(* Logix 5000 project; controller PHOTON Emulate 5570 rev 30.12; software revision 30.00; part 2 of 2 *)
(* tags used below, declared in another part *)
   PHT_Bit_indxj : DINT;
   PHT_Byte_indxi : DINT;
   PHT_D : DINT;
   PHT_Digest : DINT[60];
   PHT_DIGESTSIZE : DINT;
   PHT_GetByte_BitOffSet : DINT;
   PHT_GetByte_NoOfBits : DINT;
   PHT_GetByte_Res : DINT;
   PHT_Message : DINT[1024];
   PHT_MsgBitLen : DINT;
   PHT_Per_i : DINT;
   PHT_Per_r : DINT;
   PHT_RATEP : DINT;
   PHT_RC : DINT[8,12];
   PHT_round : DINT;
   PHT_S : DINT;
   PHT_SCS_c : DINT;
   PHT_SCS_i : DINT;
   PHT_SCS_index : DINT;
   PHT_SCS_indxi : DINT;
   PHT_SCS_j : DINT;
   PHT_SCS_OS : DINT[8,8];
   PHT_SCS_r : DINT;
   PHT_SCS_v : DINT[2];
   PHT_Squeeze_i : DINT;
   PHT_Squeeze_tmp : DINT;
   PHT_State : DINT[8,8];
   PHT_Table : DINT[8,256,2];
   PHT_Tmp : DINT[2];
   PHT_Ver : DINT;
   PHT_WordToByte_BitOffSet : DINT;
   PHT_WordToByte_i : DINT;
   PHT_WordToByte_NoOfBits : DINT;
   PHT_WordXorByte_BitOffSet : DINT;
   PHT_WordXorByte_i : DINT;
   PHT_WordXorByte_NoOfBits : DINT;
   PHT_WordXorByte_WordOffset : DINT;
   PHT_WriteByte_BitOffset : DINT;
   PHT_WriteByte_LocalFilter : DINT;
   PHT_WriteByte_NoOfBits : DINT;
   PHT_WriteByte_Value : DINT;
   Test_i : DINT;
(* MainProgram, continued *)

   		 PHT_Table[0,139,1]:=31475;
   		 PHT_Table[1,139,0]:=-1469736252;
   		 PHT_Table[1,139,1]:=18301;
   		 PHT_Table[2,139,0]:=-1123298825;
   		 PHT_Table[2,139,1]:=15795;
   		 PHT_Table[3,139,0]:=685799435;
   		 PHT_Table[3,139,1]:=31438;
   		 PHT_Table[4,139,0]:=244012053;
   		 PHT_Table[4,139,1]:=15758;
   		 PHT_Table[5,139,0]:=-1548456453;
   		 PHT_Table[5,139,1]:=62656;
   		 PHT_Table[0,140,0]:=-61122167;
   		 PHT_Table[0,140,1]:=51213;
   		 PHT_Table[1,140,0]:=-1895324903;
   		 PHT_Table[1,140,1]:=44110;
   		 PHT_Table[2,140,0]:=808429162;
   		 PHT_Table[2,140,1]:=25639;
   		 PHT_Table[3,140,0]:=-613714385;
   		 PHT_Table[3,140,1]:=51305;
   		 PHT_Table[4,140,0]:=393988799;
   		 PHT_Table[4,140,1]:=25667;
   		 PHT_Table[5,140,0]:=-1600009789;
   		 PHT_Table[5,140,1]:=35710;
   		 PHT_Table[0,141,0]:=-283086275;
   		 PHT_Table[0,141,1]:=47838;
   		 PHT_Table[1,141,0]:=-874550308;
   		 PHT_Table[1,141,1]:=59147;
   		 PHT_Table[2,141,0]:=-237246728;
   		 PHT_Table[2,141,1]:=23944;
   		 PHT_Table[3,141,0]:=1741793755;
   		 PHT_Table[3,141,1]:=47747;
   		 PHT_Table[4,141,0]:=2037901370;
   		 PHT_Table[4,141,1]:=24021;
   		 PHT_Table[5,141,0]:=272208786;
   		 PHT_Table[5,141,1]:=28666;
   		 PHT_Table[0,142,0]:=1062264297;
   		 PHT_Table[0,142,1]:=13000;
   		 PHT_Table[1,142,0]:=1699180237;
   		 PHT_Table[1,142,1]:=11166;
   		 PHT_Table[2,142,0]:=206414999;
   		 PHT_Table[2,142,1]:=6479;
   		 PHT_Table[3,142,0]:=1885114445;
   		 PHT_Table[3,142,1]:=13009;
   		 PHT_Table[4,142,0]:=1129889641;
   		 PHT_Table[4,142,1]:=6486;
   		 PHT_Table[5,142,0]:=686029174;
   		 PHT_Table[5,142,1]:=25746;
   		 PHT_Table[0,143,0]:=74596581;
   		 PHT_Table[0,143,1]:=59061;
   		 PHT_Table[1,143,0]:=-1286663590;
   		 PHT_Table[1,143,1]:=38276;
   		 PHT_Table[2,143,0]:=-2037747731;
   		 PHT_Table[2,143,1]:=29506;
   		 PHT_Table[3,143,0]:=1190447754;
   		 PHT_Table[3,143,1]:=59078;
   		 PHT_Table[4,143,0]:=-998255563;
   		 PHT_Table[4,143,1]:=29489;
   		 PHT_Table[5,143,0]:=958463749;
   		 PHT_Table[5,143,1]:=55042;
   		 PHT_Table[0,144,0]:=1954349543;
   		 PHT_Table[0,144,1]:=49197;
   		 PHT_Table[1,144,0]:=1673195800;
   		 PHT_Table[1,144,1]:=41078;
   		 PHT_Table[2,144,0]:=1288713999;
   		 PHT_Table[2,144,1]:=24635;
   		 PHT_Table[3,144,0]:=1328665040;
   		 PHT_Table[3,144,1]:=49229;
   		 PHT_Table[4,144,0]:=2013051951;
   		 PHT_Table[4,144,1]:=24667;
   		 PHT_Table[5,144,0]:=-1282539927;
   		 PHT_Table[5,144,1]:=39738;
   		 PHT_Table[0,145,0]:=-1842813959;
   		 PHT_Table[0,145,1]:=6500;
   		 PHT_Table[1,145,0]:=-1079101461;
   		 PHT_Table[1,145,1]:=38991;
   		 PHT_Table[2,145,0]:=111891142;
   		 PHT_Table[2,145,1]:=33194;
   		 PHT_Table[3,145,0]:=942557355;
   		 PHT_Table[3,145,1]:=6629;
   		 PHT_Table[4,145,0]:=-1406348615;
   		 PHT_Table[4,145,1]:=33067;
   		 PHT_Table[5,145,0]:=352121147;
   		 PHT_Table[5,145,1]:=12873;
   		 PHT_Table[0,146,0]:=-1112857175;
   		 PHT_Table[0,146,1]:=40526;
   		 PHT_Table[1,146,0]:=550375765;
   		 PHT_Table[1,146,1]:=53751;
   		 PHT_Table[2,146,0]:=620253640;
   		 PHT_Table[2,146,1]:=20470;
   		 PHT_Table[3,146,0]:=1267719672;
   		 PHT_Table[3,146,1]:=40449;
   		 PHT_Table[4,146,0]:=-762114044;
   		 PHT_Table[4,146,1]:=20409;
   		 PHT_Table[5,146,0]:=-660612775;
   		 PHT_Table[5,146,1]:=10195;
   		 PHT_Table[0,147,0]:=2097713604;
   		 PHT_Table[0,147,1]:=41914;
   		 PHT_Table[1,147,0]:=1953586231;
   		 PHT_Table[1,147,1]:=32580;
   		 PHT_Table[2,147,0]:=-143608770;
   		 PHT_Table[2,147,1]:=56354;
   		 PHT_Table[3,147,0]:=1610604912;
   		 PHT_Table[3,147,1]:=41830;
   		 PHT_Table[4,147,0]:=-715441533;
   		 PHT_Table[4,147,1]:=56574;
   		 PHT_Table[5,147,0]:=80044713;
   		 PHT_Table[5,147,1]:=23987;
   		 PHT_Table[0,148,0]:=1748556394;
   		 PHT_Table[0,148,1]:=17419;
   		 PHT_Table[1,148,0]:=1464635269;
   		 PHT_Table[1,148,1]:=26311;
   		 PHT_Table[2,148,0]:=-213179974;
   		 PHT_Table[2,148,1]:=8942;
   		 PHT_Table[3,148,0]:=-2033479349;
   		 PHT_Table[3,148,1]:=17449;
   		 PHT_Table[4,148,0]:=496674468;
   		 PHT_Table[4,148,1]:=8908;
   		 PHT_Table[5,148,0]:=476919154;
   		 PHT_Table[5,148,1]:=34868;
   		 PHT_Table[0,149,0]:=1668573878;
   		 PHT_Table[0,149,1]:=21579;
   		 PHT_Table[1,149,0]:=-1808979065;
   		 PHT_Table[1,149,1]:=32439;
   		 PHT_Table[2,149,0]:=195958896;
   		 PHT_Table[2,149,1]:=10966;
   		 PHT_Table[3,149,0]:=-1249917778;
   		 PHT_Table[3,149,1]:=21601;
   		 PHT_Table[4,149,0]:=-577811809;
   		 PHT_Table[4,149,1]:=11004;
   		 PHT_Table[5,149,0]:=976575293;
   		 PHT_Table[5,149,1]:=43196;
   		 PHT_Table[0,150,0]:=-1506505012;
   		 PHT_Table[0,150,1]:=15340;
   		 PHT_Table[1,150,0]:=428408100;
   		 PHT_Table[1,150,1]:=43937;
   		 PHT_Table[2,150,0]:=-234631269;
   		 PHT_Table[2,150,1]:=37085;
   		 PHT_Table[3,150,0]:=2076609795;
   		 PHT_Table[3,150,1]:=15228;
   		 PHT_Table[4,150,0]:=794919403;
   		 PHT_Table[4,150,1]:=36941;
   		 PHT_Table[5,150,0]:=440886786;
   		 PHT_Table[5,150,1]:=30291;
   		 PHT_Table[0,151,0]:=-1142929997;
   		 PHT_Table[0,151,1]:=2860;
   		 PHT_Table[1,151,0]:=1194002978;
   		 PHT_Table[1,151,1]:=33585;
   		 PHT_Table[2,151,0]:=-516455202;
   		 PHT_Table[2,151,1]:=34965;
   		 PHT_Table[3,151,0]:=771846711;
   		 PHT_Table[3,151,1]:=2980;
   		 PHT_Table[4,151,0]:=1952362150;
   		 PHT_Table[4,151,1]:=34845;
   		 PHT_Table[5,151,0]:=1890571475;
   		 PHT_Table[5,151,1]:=5840;
   		 PHT_Table[0,152,0]:=-1805417501;
   		 PHT_Table[0,152,1]:=35846;
   		 PHT_Table[1,152,0]:=-666162020;
   		 PHT_Table[1,152,1]:=51849;
   		 PHT_Table[2,152,0]:=-1016821808;
   		 PHT_Table[2,152,1]:=18121;
   		 PHT_Table[3,152,0]:=1570826084;
   		 PHT_Table[3,152,1]:=35904;
   		 PHT_Table[4,152,0]:=182545435;
   		 PHT_Table[4,152,1]:=18063;
   		 PHT_Table[5,152,0]:=-1127416655;
   		 PHT_Table[5,152,1]:=842;
   		 PHT_Table[0,153,0]:=61353997;
   		 PHT_Table[0,153,1]:=50993;
   		 PHT_Table[1,153,0]:=-1090551626;
   		 PHT_Table[1,153,1]:=10595;
   		 PHT_Table[2,153,0]:=-269818101;
   		 PHT_Table[2,153,1]:=61116;
   		 PHT_Table[3,153,0]:=-1085809942;
   		 PHT_Table[3,153,1]:=51167;
   		 PHT_Table[4,153,0]:=1407934289;
   		 PHT_Table[4,153,1]:=61010;
   		 PHT_Table[5,153,0]:=1410894661;
   		 PHT_Table[5,153,1]:=38284;
   		 PHT_Table[0,154,0]:=-2125215667;
   		 PHT_Table[0,154,1]:=27575;
   		 PHT_Table[1,154,0]:=-76087506;
   		 PHT_Table[1,154,1]:=54026;
   		 PHT_Table[2,154,0]:=-950070700;
   		 PHT_Table[2,154,1]:=47109;
   		 PHT_Table[3,154,0]:=-2070636705;
   		 PHT_Table[3,154,1]:=27407;
   		 PHT_Table[4,154,0]:=-1038028740;
   		 PHT_Table[4,154,1]:=47293;
   		 PHT_Table[5,154,0]:=-1536906390;
   		 PHT_Table[5,154,1]:=54989;
   		 PHT_Table[0,155,0]:=-1631706163;
   		 PHT_Table[0,155,1]:=10400;
   		 PHT_Table[1,155,0]:=1904148741;
   		 PHT_Table[1,155,1]:=15576;
   		 PHT_Table[2,155,0]:=-1758534678;
   		 PHT_Table[2,155,1]:=5228;
   		 PHT_Table[3,155,0]:=-232190674;
   		 PHT_Table[3,155,1]:=10420;
   		 PHT_Table[4,155,0]:=-72501786;
   		 PHT_Table[4,155,1]:=5240;
   		 PHT_Table[5,155,0]:=1604119348;
   		 PHT_Table[5,155,1]:=20559;
   		 PHT_Table[0,156,0]:=958119411;
   		 PHT_Table[0,156,1]:=42922;
   		 PHT_Table[1,156,0]:=44201402;
   		 PHT_Table[1,156,1]:=31064;
   		 PHT_Table[2,156,0]:=-914198143;
   		 PHT_Table[2,156,1]:=56876;
   		 PHT_Table[3,156,0]:=366100354;
   		 PHT_Table[3,156,1]:=42868;
   		 PHT_Table[4,156,0]:=-443219509;
   		 PHT_Table[4,156,1]:=57074;
   		 PHT_Table[5,156,0]:=-2133592836;
   		 PHT_Table[5,156,1]:=21905;
   		 PHT_Table[0,157,0]:=-1984477028;
   		 PHT_Table[0,157,1]:=48326;
   		 PHT_Table[1,157,0]:=-2031559782;
   		 PHT_Table[1,157,1]:=57881;
   		 PHT_Table[2,157,0]:=-800011115;
   		 PHT_Table[2,157,1]:=24193;
   		 PHT_Table[3,157,0]:=140974160;
   		 PHT_Table[3,157,1]:=48280;
   		 PHT_Table[4,157,0]:=1373520726;
   		 PHT_Table[4,157,1]:=24287;
   		 PHT_Table[5,157,0]:=-702263712;
   		 PHT_Table[5,157,1]:=25545;
   		 PHT_Table[0,158,0]:=1843104381;
   		 PHT_Table[0,158,1]:=5720;
   		 PHT_Table[1,158,0]:=-1906961340;
   		 PHT_Table[1,158,1]:=7522;
   		 PHT_Table[2,158,0]:=-647097433;
   		 PHT_Table[2,158,1]:=2865;
   		 PHT_Table[3,158,0]:=1543693422;
   		 PHT_Table[3,158,1]:=5715;
   		 PHT_Table[4,158,0]:=-390314153;
   		 PHT_Table[4,158,1]:=2874;
   		 PHT_Table[5,158,0]:=-532302915;
   		 PHT_Table[5,158,1]:=11451;
   		 PHT_Table[0,159,0]:=-1816530165;
   		 PHT_Table[0,159,1]:=44418;
   		 PHT_Table[1,159,0]:=-704922000;
   		 PHT_Table[1,159,1]:=30318;
   		 PHT_Table[2,159,0]:=-1442574538;
   		 PHT_Table[2,159,1]:=56119;
   		 PHT_Table[3,159,0]:=-1542195452;
   		 PHT_Table[3,159,1]:=44377;
   		 PHT_Table[4,159,0]:=-1653217409;
   		 PHT_Table[4,159,1]:=56300;
   		 PHT_Table[5,159,0]:=-772503311;
   		 PHT_Table[5,159,1]:=16836;
   		 PHT_Table[0,160,0]:=-992873336;
   		 PHT_Table[0,160,1]:=56129;
   		 PHT_Table[1,160,0]:=-403677384;
   		 PHT_Table[1,160,1]:=15159;
   		 PHT_Table[2,160,0]:=1426229787;
   		 PHT_Table[2,160,1]:=57494;
   		 PHT_Table[3,160,0]:=1384445442;
   		 PHT_Table[3,160,1]:=56225;
   		 PHT_Table[4,160,0]:=-1011351886;
   		 PHT_Table[4,160,1]:=57462;
   		 PHT_Table[5,160,0]:=-444971787;
   		 PHT_Table[5,160,1]:=44386;
   		 PHT_Table[0,161,0]:=2124456393;
   		 PHT_Table[0,161,1]:=25739;
   		 PHT_Table[1,161,0]:=-896607103;
   		 PHT_Table[1,161,1]:=22055;
   		 PHT_Table[2,161,0]:=412767029;
   		 PHT_Table[2,161,1]:=12958;
   		 PHT_Table[3,161,0]:=-524797030;
   		 PHT_Table[3,161,1]:=25785;
   		 PHT_Table[4,161,0]:=-2035259950;
   		 PHT_Table[4,161,1]:=12972;
   		 PHT_Table[5,161,0]:=1356720620;
   		 PHT_Table[5,161,1]:=51263;
   		 PHT_Table[0,162,0]:=1978405141;
   		 PHT_Table[0,162,1]:=29899;
   		 PHT_Table[1,162,0]:=166688899;
   		 PHT_Table[1,162,1]:=20055;
   		 PHT_Table[2,162,0]:=-528520449;
   		 PHT_Table[2,162,1]:=15014;
   		 PHT_Table[3,162,0]:=-754160001;
   		 PHT_Table[3,162,1]:=29937;
   		 PHT_Table[4,162,0]:=1185253865;
   		 PHT_Table[4,162,1]:=15004;
   		 PHT_Table[5,162,0]:=1988462499;
   		 PHT_Table[5,162,1]:=59575;
   		 PHT_Table[0,163,0]:=1331666155;
   		 PHT_Table[0,163,1]:=5200;
   		 PHT_Table[1,163,0]:=-1246589553;
   		 PHT_Table[1,163,1]:=7788;
   		 PHT_Table[2,163,0]:=-971506571;
   		 PHT_Table[2,163,1]:=2614;
   		 PHT_Table[3,163,0]:=2040105751;
   		 PHT_Table[3,163,1]:=5210;
   		 PHT_Table[4,163,0]:=-254027917;
   		 PHT_Table[4,163,1]:=2620;
   		 PHT_Table[5,163,0]:=-1571882982;
   		 PHT_Table[5,163,1]:=10410;
   		 PHT_Table[0,164,0]:=1906201072;
   		 PHT_Table[0,164,1]:=37502;
   		 PHT_Table[1,164,0]:=-1163892007;
   		 PHT_Table[1,164,1]:=56275;
   		 PHT_Table[2,164,0]:=1727333650;
   		 PHT_Table[2,164,1]:=18916;
   		 PHT_Table[3,164,0]:=-1778866955;
   		 PHT_Table[3,164,1]:=37431;
   		 PHT_Table[4,164,0]:=-2099618340;
   		 PHT_Table[4,164,1]:=18861;
   		 PHT_Table[5,164,0]:=1336244390;
   		 PHT_Table[5,164,1]:=16309;
   		 PHT_Table[0,165,0]:=-868912039;
   		 PHT_Table[0,165,1]:=3120;
   		 PHT_Table[1,165,0]:=-1704035444;
   		 PHT_Table[1,165,1]:=2596;
   		 PHT_Table[2,165,0]:=1108169946;
   		 PHT_Table[2,165,1]:=1554;
   		 PHT_Table[3,165,0]:=-562595571;
   		 PHT_Table[3,165,1]:=3126;
   		 PHT_Table[4,165,0]:=1346981336;
   		 PHT_Table[4,165,1]:=1556;
   		 PHT_Table[5,165,0]:=-1757765121;
   		 PHT_Table[5,165,1]:=6246;
   		 PHT_Table[0,166,0]:=-1542607309;
   		 PHT_Table[0,166,1]:=18491;
   		 PHT_Table[1,166,0]:=-853347319;
   		 PHT_Table[1,166,1]:=27875;
   		 PHT_Table[2,166,0]:=-1320782496;
   		 PHT_Table[2,166,1]:=9468;
   		 PHT_Table[3,166,0]:=1488775238;
   		 PHT_Table[3,166,1]:=18463;
   		 PHT_Table[4,166,0]:=1305734012;
   		 PHT_Table[4,166,1]:=9432;
   		 PHT_Table[5,166,0]:=-1957194611;
   		 PHT_Table[5,166,1]:=36946;
   		 PHT_Table[0,167,0]:=-844864341;
   		 PHT_Table[0,167,1]:=47318;
   		 PHT_Table[1,167,0]:=-264506857;
   		 PHT_Table[1,167,1]:=58373;
   		 PHT_Table[2,167,0]:=-291370710;
   		 PHT_Table[2,167,1]:=23695;
   		 PHT_Table[3,167,0]:=1112196770;
   		 PHT_Table[3,167,1]:=47242;
   		 PHT_Table[4,167,0]:=1628469278;
   		 PHT_Table[4,167,1]:=23763;
   		 PHT_Table[5,167,0]:=1379063861;
   		 PHT_Table[5,167,1]:=27627;
   		 PHT_Table[0,168,0]:=-1394004254;
   		 PHT_Table[0,168,1]:=40778;
   		 PHT_Table[1,168,0]:=-1329803075;
   		 PHT_Table[1,168,1]:=24048;
   		 PHT_Table[2,168,0]:=-1505121375;
   		 PHT_Table[2,168,1]:=49784;
   		 PHT_Table[3,168,0]:=-732993719;
   		 PHT_Table[3,168,1]:=40840;
   		 PHT_Table[4,168,0]:=-567453674;
   		 PHT_Table[4,168,1]:=49850;
   		 PHT_Table[5,168,0]:=-115904121;
   		 PHT_Table[5,168,1]:=9558;
   		 PHT_Table[0,169,0]:=-1728756777;
   		 PHT_Table[0,169,1]:=48578;
   		 PHT_Table[1,169,0]:=379198066;
   		 PHT_Table[1,169,1]:=28190;
   		 PHT_Table[2,169,0]:=1390491388;
   		 PHT_Table[2,169,1]:=54031;
   		 PHT_Table[3,169,0]:=-1750621471;
   		 PHT_Table[3,169,1]:=48401;
   		 PHT_Table[4,169,0]:=1566575428;
   		 PHT_Table[4,169,1]:=54236;
   		 PHT_Table[5,169,0]:=-139663682;
   		 PHT_Table[5,169,1]:=24908;
   		 PHT_Table[0,170,0]:=535686016;
   		 PHT_Table[0,170,1]:=17175;
   		 PHT_Table[1,170,0]:=-1979056597;
   		 PHT_Table[1,170,1]:=61394;
   		 PHT_Table[2,170,0]:=1349644734;
   		 PHT_Table[2,170,1]:=44137;
   		 PHT_Table[3,170,0]:=1992137329;
   		 PHT_Table[3,170,1]:=17339;
   		 PHT_Table[4,170,0]:=965559770;
   		 PHT_Table[4,170,1]:=44229;
   		 PHT_Table[5,170,0]:=-67616674;
   		 PHT_Table[5,170,1]:=34434;
   		 PHT_Table[0,171,0]:=812527056;
   		 PHT_Table[0,171,1]:=50237;
   		 PHT_Table[1,171,0]:=359258261;
   		 PHT_Table[1,171,1]:=42602;
   		 PHT_Table[2,171,0]:=1914892976;
   		 PHT_Table[2,171,1]:=25141;
   		 PHT_Table[3,171,0]:=85724962;
   		 PHT_Table[3,171,1]:=50271;
   		 PHT_Table[4,171,0]:=1194493799;
   		 PHT_Table[4,171,1]:=25175;
   		 PHT_Table[5,171,0]:=932931644;
   		 PHT_Table[5,171,1]:=37656;
   		 PHT_Table[0,172,0]:=-2068801446;
   		 PHT_Table[0,172,1]:=14820;
   		 PHT_Table[1,172,0]:=577529071;
   		 PHT_Table[1,172,1]:=43183;
   		 PHT_Table[2,172,0]:=-310763447;
   		 PHT_Table[2,172,1]:=37338;
   		 PHT_Table[3,172,0]:=1583211130;
   		 PHT_Table[3,172,1]:=14709;
   		 PHT_Table[4,172,0]:=923144655;
   		 PHT_Table[4,172,1]:=37195;
   		 PHT_Table[5,172,0]:=1481387429;
   		 PHT_Table[5,172,1]:=29250;
   		 PHT_Table[0,173,0]:=211206196;
   		 PHT_Table[0,173,1]:=12740;
   		 PHT_Table[1,173,0]:=-825149714;
   		 PHT_Table[1,173,1]:=42135;
   		 PHT_Table[2,173,0]:=-1853509332;
   		 PHT_Table[2,173,1]:=38342;
   		 PHT_Table[3,173,0]:=-905493115;
   		 PHT_Table[3,173,1]:=12625;
   		 PHT_Table[4,173,0]:=1468098399;
   		 PHT_Table[4,173,1]:=38227;
   		 PHT_Table[5,173,0]:=1264589327;
   		 PHT_Table[5,173,1]:=25094;
   		 PHT_Table[0,174,0]:=1291300070;
   		 PHT_Table[0,174,1]:=54113;
   		 PHT_Table[1,174,0]:=189599033;
   		 PHT_Table[1,174,1]:=14095;
   		 PHT_Table[2,174,0]:=704453502;
   		 PHT_Table[2,174,1]:=58506;
   		 PHT_Table[3,174,0]:=-958508547;
   		 PHT_Table[3,174,1]:=54149;
   		 PHT_Table[4,174,0]:=-1557100510;
   		 PHT_Table[4,174,1]:=58478;
   		 PHT_Table[5,174,0]:=-162106529;
   		 PHT_Table[5,174,1]:=48422;
   		 PHT_Table[0,175,0]:=1261296654;
   		 PHT_Table[0,175,1]:=62181;
   		 PHT_Table[1,175,0]:=117284821;
   		 PHT_Table[1,175,1]:=35816;
   		 PHT_Table[2,175,0]:=1084068760;
   		 PHT_Table[2,175,1]:=31092;
   		 PHT_Table[3,175,0]:=1064124829;
   		 PHT_Table[3,175,1]:=62108;
   		 PHT_Table[4,175,0]:=883163974;
   		 PHT_Table[4,175,1]:=30989;
   		 PHT_Table[5,175,0]:=-1687288033;
   		 PHT_Table[5,175,1]:=65448;
   		 PHT_Table[0,176,0]:=710972999;
   		 PHT_Table[0,176,1]:=54649;
   		 PHT_Table[1,176,0]:=1182449023;
   		 PHT_Table[1,176,1]:=12829;
   		 PHT_Table[2,176,0]:=141963539;
   		 PHT_Table[2,176,1]:=59267;
   		 PHT_Table[3,176,0]:=-1452744586;
   		 PHT_Table[3,176,1]:=54686;
   		 PHT_Table[4,176,0]:=-1952898226;
   		 PHT_Table[4,176,1]:=59236;
   		 PHT_Table[5,176,0]:=810266285;
   		 PHT_Table[5,176,1]:=45333;
   		 PHT_Table[0,177,0]:=-474566135;
   		 PHT_Table[0,177,1]:=35610;
   		 PHT_Table[1,177,0]:=84827442;
   		 PHT_Table[1,177,1]:=17308;
   		 PHT_Table[2,177,0]:=1616795604;
   		 PHT_Table[2,177,1]:=51278;
   		 PHT_Table[3,177,0]:=-1378423714;
   		 PHT_Table[3,177,1]:=35794;
   		 PHT_Table[4,177,0]:=787910501;
   		 PHT_Table[4,177,1]:=51334;
   		 PHT_Table[5,177,0]:=1532594589;
   		 PHT_Table[5,177,1]:=3580;
   		 PHT_Table[0,178,0]:=-738005199;
   		 PHT_Table[0,178,1]:=28323;
   		 PHT_Table[1,178,0]:=500635467;
   		 PHT_Table[1,178,1]:=22801;
   		 PHT_Table[2,178,0]:=2065444226;
   		 PHT_Table[2,178,1]:=14213;
   		 PHT_Table[3,178,0]:=1366946588;
   		 PHT_Table[3,178,1]:=28308;
   		 PHT_Table[4,178,0]:=-28277914;
   		 PHT_Table[4,178,1]:=14258;
   		 PHT_Table[5,178,0]:=33199585;
   		 PHT_Table[5,178,1]:=56426;
   		 PHT_Table[0,179,0]:=-711721021;
   		 PHT_Table[0,179,1]:=55877;
   		 PHT_Table[1,179,0]:=2005049040;
   		 PHT_Table[1,179,1]:=46896;
   		 PHT_Table[2,179,0]:=-676106126;
   		 PHT_Table[2,179,1]:=27928;
   		 PHT_Table[3,179,0]:=-851161933;
   		 PHT_Table[3,179,1]:=55848;
   		 PHT_Table[4,179,0]:=-821447008;
   		 PHT_Table[4,179,1]:=28021;
   		 PHT_Table[5,179,0]:=-990712789;
   		 PHT_Table[5,179,1]:=45031;
   		 PHT_Table[0,180,0]:=289540939;
   		 PHT_Table[0,180,1]:=260;
   		 PHT_Table[1,180,0]:=-1871527448;
   		 PHT_Table[1,180,1]:=35847;
   		 PHT_Table[2,180,0]:=-2102265239;
   		 PHT_Table[2,180,1]:=36238;
   		 PHT_Table[3,180,0]:=-1614759247;
   		 PHT_Table[3,180,1]:=393;
   		 PHT_Table[4,180,0]:=213796882;
   		 PHT_Table[4,180,1]:=36099;
   		 PHT_Table[5,180,0]:=562604254;
   		 PHT_Table[5,180,1]:=645;
   		 PHT_Table[0,181,0]:=1421883278;
   		 PHT_Table[0,181,1]:=45554;
   		 PHT_Table[1,181,0]:=-1930141186;
   		 PHT_Table[1,181,1]:=25658;
   		 PHT_Table[2,181,0]:=283927078;
   		 PHT_Table[2,181,1]:=54557;
   		 PHT_Table[3,181,0]:=1238424556;
   		 PHT_Table[3,181,1]:=45351;
   		 PHT_Table[4,181,0]:=220808860;
   		 PHT_Table[4,181,1]:=54728;
   		 PHT_Table[5,181,0]:=1620461377;
   		 PHT_Table[5,181,1]:=31018;
   		 PHT_Table[0,182,0]:=-1624296641;
   		 PHT_Table[0,182,1]:=40006;
   		 PHT_Table[1,182,0]:=455772318;
   		 PHT_Table[1,182,1]:=54009;
   		 PHT_Table[2,182,0]:=998358554;
   		 PHT_Table[2,182,1]:=20209;
   		 PHT_Table[3,182,0]:=1846850177;
   		 PHT_Table[3,182,1]:=39944;
   		 PHT_Table[4,182,0]:=-889946080;
   		 PHT_Table[4,182,1]:=20159;
   		 PHT_Table[5,182,0]:=-1701539074;
   		 PHT_Table[5,182,1]:=9154;
   		 PHT_Table[0,183,0]:=-1253071496;
   		 PHT_Table[0,183,1]:=18751;
   		 PHT_Table[1,183,0]:=1565537761;
   		 PHT_Table[1,183,1]:=57572;
   		 PHT_Table[2,183,0]:=871862025;
   		 PHT_Table[2,183,1]:=43378;
   		 PHT_Table[3,183,0]:=-948153609;
   		 PHT_Table[3,183,1]:=18838;
   		 PHT_Table[4,183,0]:=1097704302;
   		 PHT_Table[4,183,1]:=43483;
   		 PHT_Table[5,183,0]:=-1428210605;
   		 PHT_Table[5,183,1]:=37591;
   		 PHT_Table[0,184,0]:=-149427883;
   		 PHT_Table[0,184,1]:=55373;
   		 PHT_Table[1,184,0]:=1281754907;
   		 PHT_Table[1,184,1]:=46142;
   		 PHT_Table[2,184,0]:=-926244960;
   		 PHT_Table[2,184,1]:=27679;
   		 PHT_Table[3,184,0]:=-388029494;
   		 PHT_Table[3,184,1]:=55329;
   		 PHT_Table[4,184,0]:=-680647036;
   		 PHT_Table[4,184,1]:=27763;
   		 PHT_Table[5,184,0]:=-2030458996;
   		 PHT_Table[5,184,1]:=44022;
   		 PHT_Table[0,185,0]:=-2097416128;
   		 PHT_Table[0,185,1]:=44166;
   		 PHT_Table[1,185,0]:=1166639000;
   		 PHT_Table[1,185,1]:=64105;
   		 PHT_Table[2,185,0]:=683013471;
   		 PHT_Table[2,185,1]:=22201;
   		 PHT_Table[3,185,0]:=1003703733;
   		 PHT_Table[3,185,1]:=44240;
   		 PHT_Table[4,185,0]:=-1848922259;
   		 PHT_Table[4,185,1]:=22255;
   		 PHT_Table[5,185,0]:=-260300753;
   		 PHT_Table[5,185,1]:=17217;
   		 PHT_Table[0,186,0]:=1517279045;
   		 PHT_Table[0,186,1]:=62433;
   		 PHT_Table[1,186,0]:=-1768989123;
   		 PHT_Table[1,186,1]:=2031;
   		 PHT_Table[2,186,0]:=-1037276687;
   		 PHT_Table[2,186,1]:=62714;
   		 PHT_Table[3,186,0]:=-1599210708;
   		 PHT_Table[3,186,1]:=62229;
   		 PHT_Table[4,186,0]:=941247316;
   		 PHT_Table[4,186,1]:=62478;
   		 PHT_Table[5,186,0]:=-1159286847;
   		 PHT_Table[5,186,1]:=64813;
   		 PHT_Table[0,187,0]:=-1953601437;
   		 PHT_Table[0,187,1]:=53009;
   		 PHT_Table[1,187,0]:=1380111031;
   		 PHT_Table[1,187,1]:=9563;
   		 PHT_Table[2,187,0]:=-1827309970;
   		 PHT_Table[2,187,1]:=60064;
   		 PHT_Table[3,187,0]:=723352853;
   		 PHT_Table[3,187,1]:=53243;
   		 PHT_Table[4,187,0]:=862726593;
   		 PHT_Table[4,187,1]:=59978;
   		 PHT_Table[5,187,0]:=1194638575;
   		 PHT_Table[5,187,1]:=34248;
   		 PHT_Table[0,188,0]:=-555790561;
   		 PHT_Table[0,188,1]:=51717;
   		 PHT_Table[1,188,0]:=-1260176686;
   		 PHT_Table[1,188,1]:=44864;
   		 PHT_Table[2,188,0]:=794184120;
   		 PHT_Table[2,188,1]:=25888;
   		 PHT_Table[3,188,0]:=-17819306;
   		 PHT_Table[3,188,1]:=51808;
   		 PHT_Table[4,188,0]:=253516443;
   		 PHT_Table[4,188,1]:=25925;
   		 PHT_Table[5,188,0]:=-492141980;
   		 PHT_Table[5,188,1]:=36719;
   		 PHT_Table[0,189,0]:=767223471;
   		 PHT_Table[0,189,1]:=62717;
   		 PHT_Table[1,189,0]:=1271541651;
   		 PHT_Table[1,189,1]:=36602;
   		 PHT_Table[2,189,0]:=1628879349;
   		 PHT_Table[2,189,1]:=31357;
   		 PHT_Table[3,189,0]:=1356591126;
   		 PHT_Table[3,189,1]:=62599;
   		 PHT_Table[4,189,0]:=470657066;
   		 PHT_Table[4,189,1]:=31239;
   		 PHT_Table[5,189,0]:=1567873773;
   		 PHT_Table[5,189,1]:=62363;
   		 PHT_Table[0,190,0]:=1543423927;
   		 PHT_Table[0,190,1]:=18183;
   		 PHT_Table[1,190,0]:=-52766810;
   		 PHT_Table[1,190,1]:=59854;
   		 PHT_Table[2,190,0]:=1854092289;
   		 PHT_Table[2,190,1]:=44647;
   		 PHT_Table[3,190,0]:=1016087683;
   		 PHT_Table[3,190,1]:=18345;
   		 PHT_Table[4,190,0]:=155418258;
   		 PHT_Table[4,190,1]:=44745;
   		 PHT_Table[5,190,0]:=2146358795;
   		 PHT_Table[5,190,1]:=36512;
   		 PHT_Table[0,191,0]:=189575388;
   		 PHT_Table[0,191,1]:=4160;
   		 PHT_Table[1,191,0]:=-1017011198;
   		 PHT_Table[1,191,1]:=6256;
   		 PHT_Table[2,191,0]:=-119195190;
   		 PHT_Table[2,191,1]:=2104;
   		 PHT_Table[3,191,0]:=867456485;
   		 PHT_Table[3,191,1]:=4168;
   		 PHT_Table[4,191,0]:=-1072305093;
   		 PHT_Table[4,191,1]:=2096;
   		 PHT_Table[5,191,0]:=643329615;
   		 PHT_Table[5,191,1]:=8328;
   		 PHT_Table[0,192,0]:=-985602950;
   		 PHT_Table[0,192,1]:=28583;
   		 PHT_Table[1,192,0]:=-1918511453;
   		 PHT_Table[1,192,1]:=54550;
   		 PHT_Table[2,192,0]:=-106047509;
   		 PHT_Table[2,192,1]:=47627;
   		 PHT_Table[3,192,0]:=-826717779;
   		 PHT_Table[3,192,1]:=28445;
   		 PHT_Table[4,192,0]:=-219231372;
   		 PHT_Table[4,192,1]:=47793;
   		 PHT_Table[5,192,0]:=544357695;
   		 PHT_Table[5,192,1]:=57071;
   		 PHT_Table[0,193,0]:=1772735128;
   		 PHT_Table[0,193,1]:=61677;
   		 PHT_Table[1,193,0]:=1025050142;
   		 PHT_Table[1,193,1]:=35046;
   		 PHT_Table[2,193,0]:=1608809546;
   		 PHT_Table[2,193,1]:=30835;
   		 PHT_Table[3,193,0]:=452341476;
   		 PHT_Table[3,193,1]:=61589;
   		 PHT_Table[4,193,0]:=751014754;
   		 PHT_Table[4,193,1]:=30731;
   		 PHT_Table[5,193,0]:=-647672648;
   		 PHT_Table[5,193,1]:=64441;
   		 PHT_Table[0,194,0]:=-2037794651;
   		 PHT_Table[0,194,1]:=18995;
   		 PHT_Table[1,194,0]:=-154767934;
   		 PHT_Table[1,194,1]:=28653;
   		 PHT_Table[2,194,0]:=-1371563342;
   		 PHT_Table[2,194,1]:=9723;
   		 PHT_Table[3,194,0]:=2099742527;
   		 PHT_Table[3,194,1]:=18966;
   		 PHT_Table[4,194,0]:=1437891416;
   		 PHT_Table[4,194,1]:=9694;
   		 PHT_Table[5,194,0]:=-916660438;
   		 PHT_Table[5,194,1]:=37955;
   		 PHT_Table[0,195,0]:=-346934568;
   		 PHT_Table[0,195,1]:=23659;
   		 PHT_Table[1,195,0]:=2022734214;
   		 PHT_Table[1,195,1]:=29327;
   		 PHT_Table[2,195,0]:=2001832213;
   		 PHT_Table[2,195,1]:=11978;
   		 PHT_Table[3,195,0]:=556098385;
   		 PHT_Table[3,195,1]:=23621;
   		 PHT_Table[4,195,0]:=-1123533809;
   		 PHT_Table[4,195,1]:=12004;
   		 PHT_Table[5,195,0]:=689532055;
   		 PHT_Table[5,195,1]:=47352;
   		 PHT_Table[0,196,0]:=-1779264751;
   		 PHT_Table[0,196,1]:=14560;
   		 PHT_Table[1,196,0]:=-1306614521;
   		 PHT_Table[1,196,1]:=9384;
   		 PHT_Table[2,196,0]:=1875630624;
   		 PHT_Table[2,196,1]:=7252;
   		 PHT_Table[3,196,0]:=-1046652725;
   		 PHT_Table[3,196,1]:=14588;
   		 PHT_Table[4,196,0]:=1001937373;
   		 PHT_Table[4,196,1]:=7240;
   		 PHT_Table[5,196,0]:=2042922363;
   		 PHT_Table[5,196,1]:=28871;
   		 PHT_Table[0,197,0]:=1353873259;
   		 PHT_Table[0,197,1]:=22343;
   		 PHT_Table[1,197,0]:=1069249444;
   		 PHT_Table[1,197,1]:=61886;
   		 PHT_Table[2,197,0]:=-1771696693;
   		 PHT_Table[2,197,1]:=42591;
   		 PHT_Table[3,197,0]:=254021990;
   		 PHT_Table[3,197,1]:=22497;
   		 PHT_Table[4,197,0]:=-917073239;
   		 PHT_Table[4,197,1]:=42745;
   		 PHT_Table[5,197,0]:=1505146948;
   		 PHT_Table[5,197,1]:=44584;
   		 PHT_Table[0,198,0]:=37298431;
   		 PHT_Table[0,198,1]:=29655;
   		 PHT_Table[1,198,0]:=-727054035;
   		 PHT_Table[1,198,1]:=51010;
   		 PHT_Table[2,198,0]:=1128643323;
   		 PHT_Table[2,198,1]:=46113;
   		 PHT_Table[3,198,0]:=595223877;
   		 PHT_Table[3,198,1]:=29539;
   		 PHT_Table[4,198,0]:=1655859863;
   		 PHT_Table[4,198,1]:=46229;
   		 PHT_Table[5,198,0]:=-1861160305;
   		 PHT_Table[5,198,1]:=58881;
   		 PHT_Table[0,199,0]:=617576076;
   		 PHT_Table[0,199,1]:=38762;
   		 PHT_Table[1,199,0]:=1543602876;
   		 PHT_Table[1,199,1]:=20936;
   		 PHT_Table[2,199,0]:=-625591612;
   		 PHT_Table[2,199,1]:=50788;
   		 PHT_Table[3,199,0]:=1075167414;
   		 PHT_Table[3,199,1]:=38828;
   		 PHT_Table[4,199,0]:=-1096143226;
   		 PHT_Table[4,199,1]:=50850;
   		 PHT_Table[5,199,0]:=-365214163;
   		 PHT_Table[5,199,1]:=13586;
   		 PHT_Table[0,200,0]:=-811776940;
   		 PHT_Table[0,200,1]:=51969;
   		 PHT_Table[1,200,0]:=613546810;
   		 PHT_Table[1,200,1]:=9031;
   		 PHT_Table[2,200,0]:=-1377324079;
   		 PHT_Table[2,200,1]:=59566;
   		 PHT_Table[3,200,0]:=1630577639;
   		 PHT_Table[3,200,1]:=52201;
   		 PHT_Table[4,200,0]:=60953225;
   		 PHT_Table[4,200,1]:=59462;
   		 PHT_Table[5,200,0]:=-1021171014;
   		 PHT_Table[5,200,1]:=36330;
   		 PHT_Table[0,201,0]:=1603045202;
   		 PHT_Table[0,201,1]:=41394;
   		 PHT_Table[1,201,0]:=1335215612;
   		 PHT_Table[1,201,1]:=31818;
   		 PHT_Table[2,201,0]:=-402039828;
   		 PHT_Table[2,201,1]:=56613;
   		 PHT_Table[3,201,0]:=2053410313;
   		 PHT_Table[3,201,1]:=41327;
   		 PHT_Table[4,201,0]:=-851662169;
   		 PHT_Table[4,201,1]:=56824;
   		 PHT_Table[5,201,0]:=1187916046;
   		 PHT_Table[5,201,1]:=22946;
   		 PHT_Table[0,202,0]:=-356310486;
   		 PHT_Table[0,202,1]:=59533;
   		 PHT_Table[1,202,0]:=314961949;
   		 PHT_Table[1,202,1]:=40110;
   		 PHT_Table[2,202,0]:=-604056347;
   		 PHT_Table[2,202,1]:=29783;
   		 PHT_Table[3,202,0]:=-1122444034;
   		 PHT_Table[3,202,1]:=59641;
   		 PHT_Table[4,202,0]:=-1940846135;
   		 PHT_Table[4,202,1]:=29731;
   		 PHT_Table[5,202,0]:=-334424739;
   		 PHT_Table[5,202,1]:=52085;
   		 PHT_Table[0,203,0]:=-211441232;
   		 PHT_Table[0,203,1]:=16120;
   		 PHT_Table[1,203,0]:=-14084799;
   		 PHT_Table[1,203,1]:=8634;
   		 PHT_Table[2,203,0]:=1312878669;
   		 PHT_Table[2,203,1]:=8029;
   		 PHT_Table[3,203,0]:=-1372853952;
   		 PHT_Table[3,203,1]:=16103;
   		 PHT_Table[4,203,0]:=319943345;
   		 PHT_Table[4,203,1]:=8002;
   		 PHT_Table[5,203,0]:=-1076275063;
   		 PHT_Table[5,203,1]:=31988;
   		 PHT_Table[0,204,0]:=898465223;
   		 PHT_Table[0,204,1]:=38510;
   		 PHT_Table[1,204,0]:=-864861356;
   		 PHT_Table[1,204,1]:=56783;
   		 PHT_Table[2,204,0]:=1476903085;
   		 PHT_Table[2,204,1]:=19434;
   		 PHT_Table[3,204,0]:=-539657721;
   		 PHT_Table[3,204,1]:=38437;
   		 PHT_Table[4,204,0]:=-1307285868;
   		 PHT_Table[4,204,1]:=19361;
   		 PHT_Table[5,204,0]:=-877400333;
   		 PHT_Table[5,204,1]:=14231;
   		 PHT_Table[0,205,0]:=737248949;
   		 PHT_Table[0,205,1]:=24991;
   		 PHT_Table[1,205,0]:=741291236;
   		 PHT_Table[1,205,1]:=56380;
   		 PHT_Table[2,205,0]:=-1529254685;
   		 PHT_Table[2,205,1]:=48414;
   		 PHT_Table[3,205,0]:=894787545;
   		 PHT_Table[3,205,1]:=24866;
   		 PHT_Table[4,205,0]:=-1161816440;
   		 PHT_Table[4,205,1]:=48547;
   		 PHT_Table[5,205,0]:=-180103321;
   		 PHT_Table[5,205,1]:=49816;
   		 PHT_Table[0,206,0]:=-579371246;
   		 PHT_Table[0,206,1]:=3380;
   		 PHT_Table[1,206,0]:=169654884;
   		 PHT_Table[1,206,1]:=34339;
   		 PHT_Table[2,206,0]:=-1061376333;
   		 PHT_Table[2,206,1]:=35740;
   		 PHT_Table[3,206,0]:=1102562236;
   		 PHT_Table[3,206,1]:=3519;
   		 PHT_Table[4,206,0]:=1559692746;
   		 PHT_Table[4,206,1]:=35607;
   		 PHT_Table[5,206,0]:=-1229846239;
   		 PHT_Table[5,206,1]:=6883;
   		 PHT_Table[0,207,0]:=-824956;
   		 PHT_Table[0,207,1]:=3900;
   		 PHT_Table[1,207,0]:=838345647;
   		 PHT_Table[1,207,1]:=34093;
   		 PHT_Table[2,207,0]:=-540720799;
   		 PHT_Table[2,207,1]:=35483;
   		 PHT_Table[3,207,0]:=1680649413;
   		 PHT_Table[3,207,1]:=4022;
   		 PHT_Table[4,207,0]:=1150326254;
   		 PHT_Table[4,207,1]:=35345;
   		 PHT_Table[5,207,0]:=-189185402;
   		 PHT_Table[5,207,1]:=7922;
   		 PHT_Table[0,208,0]:=1659206212;
   		 PHT_Table[0,208,1]:=57517;
   		 PHT_Table[1,208,0]:=-25648612;
   		 PHT_Table[1,208,1]:=37014;
   		 PHT_Table[2,208,0]:=-1493088896;
   		 PHT_Table[2,208,1]:=28747;
   		 PHT_Table[3,208,0]:=692222721;
   		 PHT_Table[3,208,1]:=57565;
   		 PHT_Table[4,208,0]:=-321487015;
   		 PHT_Table[4,208,1]:=28731;
   		 PHT_Table[5,208,0]:=-12770569;
   		 PHT_Table[5,208,1]:=56113;
   		 PHT_Table[0,209,0]:=-37074565;
   		 PHT_Table[0,209,1]:=31979;
   		 PHT_Table[1,209,0]:=-447599998;
   		 PHT_Table[1,209,1]:=17007;
   		 PHT_Table[2,209,0]:=-1669268582;
   		 PHT_Table[2,209,1]:=16058;
   		 PHT_Table[3,209,0]:=1196870016;
   		 PHT_Table[3,209,1]:=31957;
   		 PHT_Table[4,209,0]:=639827833;
   		 PHT_Table[4,209,1]:=16004;
   		 PHT_Table[5,209,0]:=1705619465;
   		 PHT_Table[5,209,1]:=63731;
   		 PHT_Table[0,210,0]:=549271145;
   		 PHT_Table[0,210,1]:=29151;
   		 PHT_Table[1,210,0]:=-280063770;
   		 PHT_Table[1,210,1]:=50252;
   		 PHT_Table[2,210,0]:=1547457833;
   		 PHT_Table[2,210,1]:=46374;
   		 PHT_Table[3,210,0]:=115411516;
   		 PHT_Table[3,210,1]:=29034;
   		 PHT_Table[4,210,0]:=2060843699;
   		 PHT_Table[4,210,1]:=46483;
   		 PHT_Table[5,210,0]:=-753157848;
   		 PHT_Table[5,210,1]:=57872;
   		 PHT_Table[0,211,0]:=-1203210818;
   		 PHT_Table[0,211,1]:=52253;
   		 PHT_Table[1,211,0]:=-103511404;
   		 PHT_Table[1,211,1]:=43602;
   		 PHT_Table[2,211,0]:=249390037;
   		 PHT_Table[2,211,1]:=26153;
   		 PHT_Table[3,211,0]:=-1857640227;
   		 PHT_Table[3,211,1]:=52347;
   		 PHT_Table[4,211,0]:=666235383;
   		 PHT_Table[4,211,1]:=26191;
   		 PHT_Table[5,211,0]:=615997334;
   		 PHT_Table[5,211,1]:=33628;
   		 PHT_Table[0,212,0]:=1394231142;
   		 PHT_Table[0,212,1]:=36982;
   		 PHT_Table[1,212,0]:=-2126187758;
   		 PHT_Table[1,212,1]:=55517;
   		 PHT_Table[2,212,0]:=2039278272;
   		 PHT_Table[2,212,1]:=18659;
   		 PHT_Table[3,212,0]:=-1335637108;
   		 PHT_Table[3,212,1]:=36926;
   		 PHT_Table[4,212,0]:=-1698837000;
   		 PHT_Table[4,212,1]:=18603;
   		 PHT_Table[5,212,0]:=229520129;
   		 PHT_Table[5,212,1]:=15268;
   		 PHT_Table[0,213,0]:=1721186977;
   		 PHT_Table[0,213,1]:=1560;
   		 PHT_Table[1,213,0]:=1295495238;
   		 PHT_Table[1,213,1]:=1298;
   		 PHT_Table[2,213,0]:=562768493;
   		 PHT_Table[2,213,1]:=777;
   		 PHT_Table[3,213,0]:=1874243979;
   		 PHT_Table[3,213,1]:=1563;
   		 PHT_Table[4,213,0]:=682208108;
   		 PHT_Table[4,213,1]:=778;
   		 PHT_Table[5,213,0]:=-971121166;
   		 PHT_Table[5,213,1]:=3123;
   		 PHT_Table[0,214,0]:=511507314;
   		 PHT_Table[0,214,1]:=63473;
   		 PHT_Table[1,214,0]:=-530810960;
   		 PHT_Table[1,214,1]:=499;
   		 PHT_Table[2,214,0]:=-52515762;
   		 PHT_Table[2,214,1]:=63220;
   		 PHT_Table[3,214,0]:=-360700450;
   		 PHT_Table[3,214,1]:=63239;
   		 PHT_Table[4,214,0]:=148140060;
   		 PHT_Table[4,214,1]:=62978;
   		 PHT_Table[5,214,0]:=1055930772;
   		 PHT_Table[5,214,1]:=62735;
   		 PHT_Table[0,215,0]:=-948321147;
   		 PHT_Table[0,215,1]:=7280;
   		 PHT_Table[1,215,0]:=1494212494;
   		 PHT_Table[1,215,1]:=4692;
   		 PHT_Table[2,215,0]:=-1159172848;
   		 PHT_Table[2,215,1]:=3626;
   		 PHT_Table[3,215,0]:=-305976088;
   		 PHT_Table[3,215,1]:=7294;
   		 PHT_Table[4,215,0]:=-1872977437;
   		 PHT_Table[4,215,1]:=3620;
   		 PHT_Table[5,215,0]:=-1318924368;
   		 PHT_Table[5,215,1]:=14574;
   		 PHT_Table[0,216,0]:=1459165041;
   		 PHT_Table[0,216,1]:=49701;
   		 PHT_Table[1,216,0]:=1482582227;
   		 PHT_Table[1,216,1]:=41848;
   		 PHT_Table[2,216,0]:=1403640029;
   		 PHT_Table[2,216,1]:=24892;
   		 PHT_Table[3,216,0]:=1789574825;
   		 PHT_Table[3,216,1]:=49732;
   		 PHT_Table[4,216,0]:=1872440331;
   		 PHT_Table[4,216,1]:=24925;
   		 PHT_Table[5,216,0]:=-242829874;
   		 PHT_Table[5,216,1]:=40747;
   		 PHT_Table[0,217,0]:=-1877884154;
   		 PHT_Table[0,217,1]:=27315;
   		 PHT_Table[1,217,0]:=1795440326;
   		 PHT_Table[1,217,1]:=24333;
   		 PHT_Table[2,217,0]:=1173284925;
   		 PHT_Table[2,217,1]:=13707;
   		 PHT_Table[3,217,0]:=458501614;
   		 PHT_Table[3,217,1]:=27270;
   		 PHT_Table[4,217,0]:=-828458962;
   		 PHT_Table[4,217,1]:=13758;
   		 PHT_Table[5,217,0]:=-2048130124;
   		 PHT_Table[5,217,1]:=54344;
   		 PHT_Table[0,218,0]:=-1602228522;
   		 PHT_Table[0,218,1]:=44686;
   		 PHT_Table[1,218,0]:=2121131603;
   		 PHT_Table[1,218,1]:=63847;
   		 PHT_Table[2,218,0]:=936123021;
   		 PHT_Table[2,218,1]:=22462;
   		 PHT_Table[3,218,0]:=508043980;
   		 PHT_Table[3,218,1]:=44761;
   		 PHT_Table[4,218,0]:=-1985200311;
   		 PHT_Table[4,218,1]:=22505;
   		 PHT_Table[5,218,0]:=-1300796536;
   		 PHT_Table[5,218,1]:=18256;
   		 PHT_Table[0,219,0]:=-1546133797;
   		 PHT_Table[0,219,1]:=27071;
   		 PHT_Table[1,219,0]:=-1064147227;
   		 PHT_Table[1,219,1]:=53252;
   		 PHT_Table[2,219,0]:=-668533370;
   		 PHT_Table[2,219,1]:=47362;
   		 PHT_Table[3,219,0]:=-1592788954;
   		 PHT_Table[3,219,1]:=26886;
   		 PHT_Table[4,219,0]:=-632856552;
   		 PHT_Table[4,219,1]:=47547;
   		 PHT_Table[5,219,0]:=-428875571;
   		 PHT_Table[5,219,1]:=53980;
   		 PHT_Table[0,220,0]:=2090434870;
   		 PHT_Table[0,220,1]:=5980;
   		 PHT_Table[1,220,0]:=505730476;
   		 PHT_Table[1,220,1]:=37221;
   		 PHT_Table[2,220,0]:=1541401038;
   		 PHT_Table[2,220,1]:=34495;
   		 PHT_Table[3,220,0]:=-1010671905;
   		 PHT_Table[3,220,1]:=6106;
   		 PHT_Table[4,220,0]:=-469627067;
   		 PHT_Table[4,220,1]:=34361;
   		 PHT_Table[5,220,0]:=-1043522717;
   		 PHT_Table[5,220,1]:=11838;
   		 PHT_Table[0,221,0]:=-897706941;
   		 PHT_Table[0,221,1]:=39250;
   		 PHT_Table[1,221,0]:=-41197317;
   		 PHT_Table[1,221,1]:=22754;
   		 PHT_Table[2,221,0]:=-2017295924;
   		 PHT_Table[2,221,1]:=49521;
   		 PHT_Table[3,221,0]:=-1141254462;
   		 PHT_Table[3,221,1]:=39315;
   		 PHT_Table[4,221,0]:=-159059078;
   		 PHT_Table[4,221,1]:=49584;
   		 PHT_Table[5,221,0]:=1057664117;
   		 PHT_Table[5,221,1]:=10597;
   		 PHT_Table[0,222,0]:=-1216969337;
   		 PHT_Table[0,222,1]:=15080;
   		 PHT_Table[1,222,0]:=-1980089140;
   		 PHT_Table[1,222,1]:=10150;
   		 PHT_Table[2,222,0]:=1890727410;
   		 PHT_Table[2,222,1]:=7507;
   		 PHT_Table[3,222,0]:=-469354574;
   		 PHT_Table[3,222,1]:=15093;
   		 PHT_Table[4,222,0]:=601868793;
   		 PHT_Table[4,222,1]:=7502;
   		 PHT_Table[5,222,0]:=1003474652;
   		 PHT_Table[5,222,1]:=29910;
   		 PHT_Table[0,223,0]:=1632455241;
   		 PHT_Table[0,223,1]:=10140;
   		 PHT_Table[1,223,0]:=1082598058;
   		 PHT_Table[1,223,1]:=47605;
   		 PHT_Table[2,223,0]:=1223402123;
   		 PHT_Table[2,223,1]:=40695;
   		 PHT_Table[3,223,0]:=-1778015765;
   		 PHT_Table[3,223,1]:=9986;
   		 PHT_Table[4,223,0]:=-1086513144;
   		 PHT_Table[4,223,1]:=40553;
   		 PHT_Table[5,223,0]:=-1423595086;
   		 PHT_Table[5,223,1]:=20157;
   		 PHT_Table[0,224,0]:=-430579170;
   		 PHT_Table[0,224,1]:=55625;
   		 PHT_Table[1,224,0]:=-602618125;
   		 PHT_Table[1,224,1]:=14393;
   		 PHT_Table[2,224,0]:=1249600969;
   		 PHT_Table[2,224,1]:=57745;
   		 PHT_Table[3,224,0]:=1998559611;
   		 PHT_Table[3,224,1]:=55720;
   		 PHT_Table[4,224,0]:=-607097194;
   		 PHT_Table[4,224,1]:=57712;
   		 PHT_Table[5,224,0]:=-1485762734;
   		 PHT_Table[5,224,1]:=43379;
   		 PHT_Table[0,225,0]:=-653967369;
   		 PHT_Table[0,225,1]:=60289;
   		 PHT_Table[1,225,0]:=-1185699778;
   		 PHT_Table[1,225,1]:=5031;
   		 PHT_Table[2,225,0]:=1177993566;
   		 PHT_Table[2,225,1]:=63710;
   		 PHT_Table[3,225,0]:=121833782;
   		 PHT_Table[3,225,1]:=60281;
   		 PHT_Table[4,225,0]:=-1735863809;
   		 PHT_Table[4,225,1]:=63526;
   		 PHT_Table[5,225,0]:=-1886194140;
   		 PHT_Table[5,225,1]:=52705;
   		 PHT_Table[0,226,0]:=-1384628720;
   		 PHT_Table[0,226,1]:=11180;
   		 PHT_Table[1,226,0]:=-622241498;
   		 PHT_Table[1,226,1]:=46033;
   		 PHT_Table[2,226,0]:=182908497;
   		 PHT_Table[2,226,1]:=39141;
   		 PHT_Table[3,226,0]:=1215486182;
   		 PHT_Table[3,226,1]:=11060;
   		 PHT_Table[4,226,0]:=-277582384;
   		 PHT_Table[4,226,1]:=39037;
   		 PHT_Table[5,226,0]:=1008666701;
   		 PHT_Table[5,226,1]:=22235;
   		 PHT_Table[0,227,0]:=874278197;
   		 PHT_Table[0,227,1]:=8840;
   		 PHT_Table[1,227,0]:=-1507407153;
   		 PHT_Table[1,227,1]:=13294;
   		 PHT_Table[2,227,0]:=-190276259;
   		 PHT_Table[2,227,1]:=4471;
   		 PHT_Table[3,227,0]:=1139328424;
   		 PHT_Table[3,227,1]:=8857;
   		 PHT_Table[4,227,0]:=-2092084398;
   		 PHT_Table[4,227,1]:=4454;
   		 PHT_Table[5,227,0]:=247174969;
   		 PHT_Table[5,227,1]:=17434;
   		 PHT_Table[0,228,0]:=1572186029;
   		 PHT_Table[0,228,1]:=53861;
   		 PHT_Table[1,228,0]:=-1690317615;
   		 PHT_Table[1,228,1]:=47880;
   		 PHT_Table[2,228,0]:=-1421025001;
   		 PHT_Table[2,228,1]:=26884;
   		 PHT_Table[3,228,0]:=1495198540;
   		 PHT_Table[3,228,1]:=53772;
   		 PHT_Table[4,228,0]:=-1349599184;
   		 PHT_Table[4,228,1]:=26989;
   		 PHT_Table[5,228,0]:=-673260671;
   		 PHT_Table[5,228,1]:=49059;
   		 PHT_Table[0,229,0]:=-676667588;
   		 PHT_Table[0,229,1]:=43410;
   		 PHT_Table[1,229,0]:=-1557620739;
   		 PHT_Table[1,229,1]:=28786;
   		 PHT_Table[2,229,0]:=-1795765623;
   		 PHT_Table[2,229,1]:=55609;
   		 PHT_Table[3,229,0]:=-297915914;
   		 PHT_Table[3,229,1]:=43339;
   		 PHT_Table[4,229,0]:=-1380197321;
   		 PHT_Table[4,229,1]:=55776;
   		 PHT_Table[5,229,0]:=1440882340;
   		 PHT_Table[5,229,1]:=18918;
   		 PHT_Table[0,230,0]:=2010460650;
   		 PHT_Table[0,230,1]:=1820;
   		 PHT_Table[1,230,0]:=-582651474;
   		 PHT_Table[1,230,1]:=35093;
   		 PHT_Table[2,230,0]:=-1556426748;
   		 PHT_Table[2,230,1]:=36487;
   		 PHT_Table[3,230,0]:=-260699334;
   		 PHT_Table[3,230,1]:=1938;
   		 PHT_Table[4,230,0]:=605545342;
   		 PHT_Table[4,230,1]:=36361;
   		 PHT_Table[5,230,0]:=-409635540;
   		 PHT_Table[5,230,1]:=3766;
   		 PHT_Table[0,231,0]:=772986530;
   		 PHT_Table[0,231,1]:=13260;
   		 PHT_Table[1,231,0]:=-181031131;
   		 PHT_Table[1,231,1]:=42905;
   		 PHT_Table[2,231,0]:=-1896063234;
   		 PHT_Table[2,231,1]:=38081;
   		 PHT_Table[3,231,0]:=-274978052;
   		 PHT_Table[3,231,1]:=13144;
   		 PHT_Table[4,231,0]:=1340536699;
   		 PHT_Table[4,231,1]:=37973;
   		 PHT_Table[5,231,0]:=158028200;
   		 PHT_Table[5,231,1]:=26135;
   		 PHT_Table[0,232,0]:=-873528143;
   		 PHT_Table[0,232,1]:=11700;
   		 PHT_Table[1,232,0]:=-1746998944;
   		 PHT_Table[1,232,1]:=46787;
   		 PHT_Table[2,232,0]:=728620092;
   		 PHT_Table[2,232,1]:=39916;
   		 PHT_Table[3,232,0]:=667183469;
   		 PHT_Table[3,232,1]:=11567;
   		 PHT_Table[4,232,0]:=-941766980;
   		 PHT_Table[4,232,1]:=39799;
   		 PHT_Table[5,232,0]:=-100477505;
   		 PHT_Table[5,232,1]:=23272;
   		 PHT_Table[0,233,0]:=-773734618;
   		 PHT_Table[0,233,1]:=15600;
   		 PHT_Table[1,233,0]:=-993162102;
   		 PHT_Table[1,233,1]:=8884;
   		 PHT_Table[2,233,0]:=1362698143;
   		 PHT_Table[2,233,1]:=7770;
   		 PHT_Table[3,233,0]:=-1951365575;
   		 PHT_Table[3,233,1]:=15598;
   		 PHT_Table[4,233,0]:=192307861;
   		 PHT_Table[4,233,1]:=7748;
   		 PHT_Table[5,233,0]:=-36564178;
   		 PHT_Table[5,233,1]:=30949;
   		 PHT_Table[0,234,0]:=1578997664;
   		 PHT_Table[0,234,1]:=5460;
   		 PHT_Table[1,234,0]:=633359463;
   		 PHT_Table[1,234,1]:=37483;
   		 PHT_Table[2,234,0]:=1151731228;
   		 PHT_Table[2,234,1]:=34744;
   		 PHT_Table[3,234,0]:=-430362202;
   		 PHT_Table[3,234,1]:=5587;
   		 PHT_Table[4,234,0]:=-60448927;
   		 PHT_Table[4,234,1]:=34623;
   		 PHT_Table[5,234,0]:=-2084155196;
   		 PHT_Table[5,234,1]:=10799;
   		 PHT_Table[0,235,0]:=-317107518;
   		 PHT_Table[0,235,1]:=51465;
   		 PHT_Table[1,235,0]:=527786737;
   		 PHT_Table[1,235,1]:=8265;
   		 PHT_Table[2,235,0]:=-1298244605;
   		 PHT_Table[2,235,1]:=59817;
   		 PHT_Table[3,235,0]:=1152109726;
   		 PHT_Table[3,235,1]:=51680;
   		 PHT_Table[4,235,0]:=465928877;
   		 PHT_Table[4,235,1]:=59712;
   		 PHT_Table[5,235,0]:=-2127994595;
   		 PHT_Table[5,235,1]:=35323;
   		 PHT_Table[0,236,0]:=797165136;
   		 PHT_Table[0,236,1]:=34602;
   		 PHT_Table[1,236,0]:=-1621088578;
   		 PHT_Table[1,236,1]:=18872;
   		 PHT_Table[2,236,0]:=575865614;
   		 PHT_Table[2,236,1]:=52828;
   		 PHT_Table[3,236,0]:=1939969363;
   		 PHT_Table[3,236,1]:=34788;
   		 PHT_Table[4,236,0]:=2126496445;
   		 PHT_Table[4,236,1]:=52882;
   		 PHT_Table[5,236,0]:=-865916830;
   		 PHT_Table[5,236,1]:=5530;
   		 PHT_Table[0,237,0]:=-462634271;
   		 PHT_Table[0,237,1]:=43678;
   		 PHT_Table[1,237,0]:=146722782;
   		 PHT_Table[1,237,1]:=65403;
   		 PHT_Table[2,237,0]:=155115314;
   		 PHT_Table[2,237,1]:=21936;
   		 PHT_Table[3,237,0]:=1415969854;
   		 PHT_Table[3,237,1]:=43723;
   		 PHT_Table[4,237,0]:=-1184758783;
   		 PHT_Table[4,237,1]:=21989;
   		 PHT_Table[5,237,0]:=912391645;
   		 PHT_Table[5,237,1]:=20338;
   		 PHT_Table[0,238,0]:=661079681;
   		 PHT_Table[0,238,1]:=20571;
   		 PHT_Table[1,238,0]:=-486669814;
   		 PHT_Table[1,238,1]:=30891;
   		 PHT_Table[2,238,0]:=895278543;
   		 PHT_Table[2,238,1]:=10456;
   		 PHT_Table[3,238,0]:=-11396516;
   		 PHT_Table[3,238,1]:=20595;
   		 PHT_Table[4,238,0]:=-314478121;
   		 PHT_Table[4,238,1]:=10480;
   		 PHT_Table[5,238,0]:=-1104949912;
   		 PHT_Table[5,238,1]:=41118;
   		 PHT_Table[0,239,0]:=463448933;
   		 PHT_Table[0,239,1]:=42402;
   		 PHT_Table[1,239,0]:=960949361;
   		 PHT_Table[1,239,1]:=31318;
   		 PHT_Table[2,239,0]:=-688153005;
   		 PHT_Table[2,239,1]:=57131;
   		 PHT_Table[3,239,0]:=810111227;
   		 PHT_Table[3,239,1]:=42365;
   		 PHT_Table[4,239,0]:=-34434577;
   		 PHT_Table[4,239,1]:=57332;
   		 PHT_Table[5,239,0]:=-1025982629;
   		 PHT_Table[5,239,1]:=20864;
   		 PHT_Table[0,240,0]:=868621789;
   		 PHT_Table[0,240,1]:=780;
   		 PHT_Table[1,240,0]:=-1416210397;
   		 PHT_Table[1,240,1]:=36617;
   		 PHT_Table[2,240,0]:=-1647831621;
   		 PHT_Table[2,240,1]:=35977;
   		 PHT_Table[3,240,0]:=-1168386616;
   		 PHT_Table[3,240,1]:=896;
   		 PHT_Table[4,240,0]:=349820982;
   		 PHT_Table[4,240,1]:=35845;
   		 PHT_Table[5,240,0]:=1669587833;
   		 PHT_Table[5,240,1]:=1684;
   		 PHT_Table[0,241,0]:=-1107094108;
   		 PHT_Table[0,241,1]:=22911;
   		 PHT_Table[1,241,0]:=-1640918557;
   		 PHT_Table[1,241,1]:=63636;
   		 PHT_Table[2,241,0]:=-887966013;
   		 PHT_Table[2,241,1]:=41290;
   		 PHT_Table[3,241,0]:=-188217582;
   		 PHT_Table[3,241,1]:=23006;
   		 PHT_Table[4,241,0]:=-2122821803;
   		 PHT_Table[4,241,1]:=41451;
   		 PHT_Table[5,241,0]:=-1937288676;
   		 PHT_Table[5,241,1]:=45663;
   		 PHT_Table[0,242,0]:=-1721478363;
   		 PHT_Table[0,242,1]:=2340;
   		 PHT_Table[1,242,0]:=2093978601;
   		 PHT_Table[1,242,1]:=32831;
   		 PHT_Table[2,242,0]:=-28415220;
   		 PHT_Table[2,242,1]:=35218;
   		 PHT_Table[3,242,0]:=194649422;
   		 PHT_Table[3,242,1]:=2477;
   		 PHT_Table[4,242,0]:=1815690882;
   		 PHT_Table[4,242,1]:=35099;
   		 PHT_Table[5,242,0]:=849649524;
   		 PHT_Table[5,242,1]:=4801;
   		 PHT_Table[0,243,0]:=-1578172892;
   		 PHT_Table[0,243,1]:=6760;
   		 PHT_Table[1,243,0]:=339242952;
   		 PHT_Table[1,243,1]:=5958;
   		 PHT_Table[2,243,0]:=-1687992451;
   		 PHT_Table[2,243,1]:=3363;
   		 PHT_Table[3,243,0]:=-2106221213;
   		 PHT_Table[3,243,1]:=6757;
   		 PHT_Table[4,243,0]:=-1191900529;
   		 PHT_Table[4,243,1]:=3374;
   		 PHT_Table[5,243,0]:=2004816450;
   		 PHT_Table[5,243,1]:=13533;
   		 PHT_Table[0,244,0]:=1877125762;
   		 PHT_Table[0,244,1]:=25999;
   		 PHT_Table[1,244,0]:=1526472041;
   		 PHT_Table[1,244,1]:=55840;
   		 PHT_Table[2,244,0]:=-1708414628;
   		 PHT_Table[2,244,1]:=48912;
   		 PHT_Table[3,244,0]:=2138603819;
   		 PHT_Table[3,244,1]:=25904;
   		 PHT_Table[4,244,0]:=-1978782272;
   		 PHT_Table[4,244,1]:=49071;
   		 PHT_Table[5,244,0]:=1901412658;
   		 PHT_Table[5,244,1]:=51898;
   		 PHT_Table[0,245,0]:=149192913;
   		 PHT_Table[0,245,1]:=55153;
   		 PHT_Table[1,245,0]:=2107516084;
   		 PHT_Table[1,245,1]:=12563;
   		 PHT_Table[2,245,0]:=386916033;
   		 PHT_Table[2,245,1]:=59012;
   		 PHT_Table[3,245,0]:=-1930195185;
   		 PHT_Table[3,245,1]:=55191;
   		 PHT_Table[4,245,0]:=-1812024470;
   		 PHT_Table[4,245,1]:=58978;
   		 PHT_Table[5,245,0]:=1916855562;
   		 PHT_Table[5,245,1]:=46340;
   		 PHT_Table[0,246,0]:=474340237;
   		 PHT_Table[0,246,1]:=33830;
   		 PHT_Table[1,246,0]:=888569501;
   		 PHT_Table[1,246,1]:=50865;
   		 PHT_Table[2,246,0]:=-1080355147;
   		 PHT_Table[2,246,1]:=17109;
   		 PHT_Table[3,246,0]:=-906346341;
   		 PHT_Table[3,246,1]:=33892;
   		 PHT_Table[4,246,0]:=1785076363;
   		 PHT_Table[4,246,1]:=17047;
   		 PHT_Table[5,246,0]:=-1344222437;
   		 PHT_Table[5,246,1]:=4878;
   		 PHT_Table[0,247,0]:=2133963067;
   		 PHT_Table[0,247,1]:=53357;
   		 PHT_Table[1,247,0]:=-1596238566;
   		 PHT_Table[1,247,1]:=47110;
   		 PHT_Table[2,247,0]:=-1271591227;
   		 PHT_Table[2,247,1]:=26627;
   		 PHT_Table[3,247,0]:=2089124917;
   		 PHT_Table[3,247,1]:=53253;
   		 PHT_Table[4,247,0]:=-1209446380;
   		 PHT_Table[4,247,1]:=26731;
   		 PHT_Table[5,247,0]:=-1781166042;
   		 PHT_Table[5,247,1]:=48050;
   		 PHT_Table[0,248,0]:=2060640556;
   		 PHT_Table[0,248,1]:=33342;
   		 PHT_Table[1,248,0]:=2042744539;
   		 PHT_Table[1,248,1]:=50083;
   		 PHT_Table[2,248,0]:=-1643103016;
   		 PHT_Table[2,248,1]:=16860;
   		 PHT_Table[3,248,0]:=-1504906992;
   		 PHT_Table[3,248,1]:=33407;
   		 PHT_Table[4,248,0]:=1120907751;
   		 PHT_Table[4,248,1]:=16797;
   		 PHT_Table[5,248,0]:=1778194153;
   		 PHT_Table[5,248,1]:=7997;
   		 PHT_Table[0,249,0]:=-1879299962;
   		 PHT_Table[0,249,1]:=10660;
   		 PHT_Table[1,249,0]:=-519192339;
   		 PHT_Table[1,249,1]:=45279;
   		 PHT_Table[2,249,0]:=362748291;
   		 PHT_Table[2,249,1]:=39394;
   		 PHT_Table[3,249,0]:=1844033439;
   		 PHT_Table[3,249,1]:=10557;
   		 PHT_Table[4,249,0]:=-149684748;
   		 PHT_Table[4,249,1]:=39291;
   		 PHT_Table[5,249,0]:=2115257322;
   		 PHT_Table[5,249,1]:=21194;
   		 PHT_Table[0,250,0]:=-1916467079;
   		 PHT_Table[0,250,1]:=23155;
   		 PHT_Table[1,250,0]:=900188608;
   		 PHT_Table[1,250,1]:=30621;
   		 PHT_Table[2,250,0]:=1457169272;
   		 PHT_Table[2,250,1]:=11715;
   		 PHT_Table[3,250,0]:=1318310618;
   		 PHT_Table[3,250,1]:=23134;
   		 PHT_Table[4,250,0]:=-1784572061;
   		 PHT_Table[4,250,1]:=11758;
   		 PHT_Table[5,250,0]:=-284905115;
   		 PHT_Table[5,250,1]:=46283;
   		 PHT_Table[0,251,0]:=-436350445;
   		 PHT_Table[0,251,1]:=7800;
   		 PHT_Table[1,251,0]:=1659586117;
   		 PHT_Table[1,251,1]:=4442;
   		 PHT_Table[2,251,0]:=-1517190462;
   		 PHT_Table[2,251,1]:=3885;
   		 PHT_Table[3,251,0]:=-933739631;
   		 PHT_Table[3,251,1]:=7799;
   		 PHT_Table[4,251,0]:=-2009386553;
   		 PHT_Table[4,251,1]:=3874;
   		 PHT_Table[5,251,0]:=-211188713;
   		 PHT_Table[5,251,1]:=15615;
   		 PHT_Table[0,252,0]:=-1977649007;
   		 PHT_Table[0,252,1]:=31735;
   		 PHT_Table[1,252,0]:=941054764;
   		 PHT_Table[1,252,1]:=52090;
   		 PHT_Table[2,252,0]:=1069165470;
   		 PHT_Table[2,252,1]:=45117;
   		 PHT_Table[3,252,0]:=-1222589766;
   		 PHT_Table[3,252,1]:=31559;
   		 PHT_Table[4,252,0]:=37035015;
   		 PHT_Table[4,252,1]:=45197;
   		 PHT_Table[5,252,0]:=-2109946587;
   		 PHT_Table[5,252,1]:=63045;
   		 PHT_Table[0,253,0]:=-957819785;
   		 PHT_Table[0,253,1]:=43158;
   		 PHT_Table[1,253,0]:=861558293;
   		 PHT_Table[1,253,1]:=64629;
   		 PHT_Table[2,253,0]:=373764320;
   		 PHT_Table[2,253,1]:=21687;
   		 PHT_Table[3,253,0]:=1912509255;
   		 PHT_Table[3,253,1]:=43202;
   		 PHT_Table[4,253,0]:=-1593469915;
   		 PHT_Table[4,253,1]:=21731;
   		 PHT_Table[5,253,0]:=1953150586;
   		 PHT_Table[5,253,1]:=19299;
   		 PHT_Table[0,254,0]:=-406523156;
   		 PHT_Table[0,254,1]:=28079;
   		 PHT_Table[1,254,0]:=-1237233816;
   		 PHT_Table[1,254,1]:=54808;
   		 PHT_Table[2,254,0]:=-422299591;
   		 PHT_Table[2,254,1]:=47884;
   		 PHT_Table[3,254,0]:=-350083372;
   		 PHT_Table[3,254,1]:=27924;
   		 PHT_Table[4,254,0]:=-360096944;
   		 PHT_Table[4,254,1]:=48055;
   		 PHT_Table[5,254,0]:=1652127384;
   		 PHT_Table[5,254,1]:=56062;
   		 PHT_Table[0,255,0]:=-626192390;
   		 PHT_Table[0,255,1]:=11440;
   		 PHT_Table[1,255,0]:=128723080;
   		 PHT_Table[1,255,1]:=15044;
   		 PHT_Table[2,255,0]:=-1445190059;
   		 PHT_Table[2,255,1]:=5730;
   		 PHT_Table[3,255,0]:=-1207643172;
   		 PHT_Table[3,255,1]:=11430;
   		 PHT_Table[4,255,0]:=-882667858;
   		 PHT_Table[4,255,1]:=5748;
   		 PHT_Table[5,255,0]:=-611680927;
   		 PHT_Table[5,255,1]:=22637;
   End_CASE;
END_ROUTINE

ROUTINE PHOTON_Permutation   (* structured text *)
   
   for PHT_Per_r:=0 to PHT_round-1 by 1 do
   
   	//addkey
   	for PHT_Per_i:=0 to PHT_D-1 by 1 do
   		PHT_State[PHT_Per_i,0]:= PHT_State[PHT_Per_i,0] XOR PHT_RC[PHT_Per_i,PHT_Per_r];
   
   	end_for;
   
   	JSR(PHOTON_SCShRMCS);
   
   end_for;
END_ROUTINE

ROUTINE PHOTON_SCShRMCS   (* structured text *)
   (*
   void SCShRMCS(byte state[D][D])
   {
   	int c,r;
   	tword v;
   	byte os[D][D];
   	memcpy(os, state, D*D);
   
   	for(c = 0; c < D; c++){ // for all columns
   		v = 0;
   		for(r = 0; r < D; r++) // for all rows in this column i after ShiftRow
   			v ^= Table[r][os[r][(r+c)%D]];
   
   		for(r = 1; r <= D; r++){
   			state[D-r][c] = (byte)v & WORDFILTER;
   			v >>= S;
   		}
   	}
   }
   *)
   
   FOR PHT_SCS_i:=0 to PHT_D-1 by 1 do
   	FOR PHT_SCS_j:=0 to PHT_D-1 by 1 do
   		PHT_SCS_OS[PHT_SCS_i,PHT_SCS_j]:=PHT_State[PHT_SCS_i,PHT_SCS_j];
   	END_FOR;
   END_FOR;
   
   if PHT_Ver<=4 then
   
   	for PHT_SCS_c:= 0 to PHT_D-1 by 1 do
   		PHT_SCS_v[0]:=0;
   
   		for PHT_SCS_r:=0 to PHT_D-1 by 1 do
   			PHT_SCS_index:=PHT_SCS_OS[PHT_SCS_r,(PHT_SCS_r+PHT_SCS_c) mod PHT_D];
   			PHT_SCS_v[0]:=PHT_SCS_v[0] XOR PHT_Table[PHT_SCS_r,PHT_SCS_index,0];
   		end_for;
   
   		PHT_SCS_j:=0;
   
   		for PHT_SCS_r:=1 to PHT_D by 1 do
   			 PHT_SCS_indxi:=PHT_D-PHT_SCS_r;
   			 PHT_State[PHT_SCS_indxi,PHT_SCS_c]:=0;
   			 PHT_State[PHT_SCS_indxi,PHT_SCS_c].[0]:=PHT_SCS_v[0].[PHT_SCS_j];
   			 PHT_State[PHT_SCS_indxi,PHT_SCS_c].[1]:=PHT_SCS_v[0].[PHT_SCS_j+1];
   			 PHT_State[PHT_SCS_indxi,PHT_SCS_c].[2]:=PHT_SCS_v[0].[PHT_SCS_j+2];
   			 PHT_State[PHT_SCS_indxi,PHT_SCS_c].[3]:=PHT_SCS_v[0].[PHT_SCS_j+3];
   			 PHT_SCS_j:=PHT_SCS_j + 4;
   
   		end_for;
   	end_for;
   
   
   
    else
   
   	for PHT_SCS_c:= 0 to PHT_D-1 by 1 do
   		PHT_SCS_v[0]:=0;
   		PHT_SCS_v[1]:=0;
   
   		for PHT_SCS_r:=0 to PHT_D-1 by 1 do
   			PHT_SCS_index:=PHT_SCS_OS[PHT_SCS_r,(PHT_SCS_r+PHT_SCS_c) mod PHT_D];
   			PHT_SCS_v[0]:=PHT_SCS_v[0] XOR PHT_Table[PHT_SCS_r,PHT_SCS_index,0];
   			PHT_SCS_v[1]:=PHT_SCS_v[1] XOR PHT_Table[PHT_SCS_r,PHT_SCS_index,1];
   		end_for;
   
   		PHT_SCS_j:=0;
   		PHT_SCS_i:=0;
   
   		for PHT_SCS_r:=1 to PHT_D by 1 do
   				PHT_SCS_indxi:=PHT_D-PHT_SCS_r;
   				PHT_State[PHT_SCS_indxi,PHT_SCS_c]:=0;
   			if PHT_SCS_j < 32 then
   				PHT_State[PHT_SCS_indxi,PHT_SCS_c].[0]:=PHT_SCS_v[0].[PHT_SCS_j];
   				PHT_State[PHT_SCS_indxi,PHT_SCS_c].[1]:=PHT_SCS_v[0].[PHT_SCS_j+1];
   				PHT_State[PHT_SCS_indxi,PHT_SCS_c].[2]:=PHT_SCS_v[0].[PHT_SCS_j+2];
   				PHT_State[PHT_SCS_indxi,PHT_SCS_c].[3]:=PHT_SCS_v[0].[PHT_SCS_j+3];
   				PHT_State[PHT_SCS_indxi,PHT_SCS_c].[4]:=PHT_SCS_v[0].[PHT_SCS_j+4];
   				PHT_State[PHT_SCS_indxi,PHT_SCS_c].[5]:=PHT_SCS_v[0].[PHT_SCS_j+5];
   				PHT_State[PHT_SCS_indxi,PHT_SCS_c].[6]:=PHT_SCS_v[0].[PHT_SCS_j+6];
   				PHT_State[PHT_SCS_indxi,PHT_SCS_c].[7]:=PHT_SCS_v[0].[PHT_SCS_j+7];
   				PHT_SCS_j:=PHT_SCS_j + 8;
   
   			else
   				PHT_State[PHT_SCS_indxi,PHT_SCS_c].[0]:=PHT_SCS_v[1].[PHT_SCS_i];
   				PHT_State[PHT_SCS_indxi,PHT_SCS_c].[1]:=PHT_SCS_v[1].[PHT_SCS_i+1];
   				PHT_State[PHT_SCS_indxi,PHT_SCS_c].[2]:=PHT_SCS_v[1].[PHT_SCS_i+2];
   				PHT_State[PHT_SCS_indxi,PHT_SCS_c].[3]:=PHT_SCS_v[1].[PHT_SCS_i+3];
   				PHT_State[PHT_SCS_indxi,PHT_SCS_c].[4]:=PHT_SCS_v[1].[PHT_SCS_i+4];
   				PHT_State[PHT_SCS_indxi,PHT_SCS_c].[5]:=PHT_SCS_v[1].[PHT_SCS_i+5];
   				PHT_State[PHT_SCS_indxi,PHT_SCS_c].[6]:=PHT_SCS_v[1].[PHT_SCS_i+6];
   				PHT_State[PHT_SCS_indxi,PHT_SCS_c].[7]:=PHT_SCS_v[1].[PHT_SCS_i+7];
   				PHT_SCS_i:=PHT_SCS_i + 8;
   			end_if;
   	   end_for;
   
   	end_for;
   
   end_if;
   
END_ROUTINE

ROUTINE PHOTON_Squeeze   (* structured text *)
   (*
   void Squeeze(byte state[D][D], byte*digest)
   {
   	int i = 0;
   	while(1){
   
   		WordToByte(state, digest, i, min(RATEP, DIGESTSIZE-i));
   		i += RATEP;
   		if(i >= DIGESTSIZE) break;
   		Permutation(state, ROUND);
   	}
   }
   *)
   
   PHT_Squeeze_i:=0;
   
   PHT_Squeeze_tmp:=2;
   while PHT_Squeeze_tmp>1 do
   
   	PHT_WordToByte_BitOffSet:= PHT_Squeeze_i;
   	PHT_WordToByte_NoOfBits:= PHT_DIGESTSIZE-PHT_Squeeze_i;
   	if PHT_WordToByte_NoOfBits > PHT_RATEP then
   		PHT_WordToByte_NoOfBits:= PHT_RATEP;
   	end_if;
   	JSR(PHOTON_WordToByte);
   
   	PHT_Squeeze_i:=PHT_Squeeze_i+PHT_RATEP;
   
   	if PHT_Squeeze_i >= PHT_DIGESTSIZE then
   		exit;
   	end_if;
   
   	JSR(PHOTON_Permutation);
   end_while;
END_ROUTINE

ROUTINE PHOTON_Test   (* structured text *)
   (*
   if S:FS Then
   	PHT_Ver:=5;
   
   	PHT_BitLen:=40;
   
   	for Test_i:=0 to PHT_BitLen/8-1 by 1 do
   		PHT_Msg[Test_i]:=0;
   	end_for;
   
   	JSR(PHOTON);
   end_if;
   *)
   
   
   
   if S:FS Then
   	PHT_Ver:=0;
   
   	PHT_MsgBitLen:=8;
   
   	for Test_i:=0 to PHT_MsgBitLen/8-1 by 1 do
   		PHT_Message[Test_i]:=48;
   	end_for;
   
   
   	JSR(PHOTON);
   end_if;
   
   
END_ROUTINE

ROUTINE PHOTON_WordToByte   (* structured text *)
   (*
   void WordToByte(byte state[D][D], byte*str, int BitOffSet, int NoOfBits)
   {
   	int i = 0;
   	while(i < NoOfBits)
   	{
   		WriteByte(str, (state[i/(S*D)][(i/S)%D] & WORDFILTER)>>(S-min(S, NoOfBits-i)), BitOffSet+i, min(S, NoOfBits-i));
   		i += S;
   	});
   }
   *)
   
   // str:   PHT_Digest
   
   
   PHT_WordToByte_i:=0;
   While PHT_WordToByte_i<PHT_WordToByte_NoOfBits Do
   
   
   	//BitOffSet+i
   	PHT_WriteByte_BitOffset:=PHT_WordToByte_BitOffSet+PHT_WordToByte_i;
   	//min(S, NoOfBits-i)
   	PHT_WriteByte_NoOfBits:= PHT_WordToByte_NoOfBits - PHT_WordToByte_i;
   	if PHT_WriteByte_NoOfBits> PHT_S Then
   		PHT_WriteByte_NoOfBits:=PHT_S;
   	End_If;
   
   	PHT_Tmp[1]:=PHT_S-PHT_WriteByte_NoOfBits;
   
   	//  i/(S*D)
   	PHT_Byte_indxi:=  PHT_WordToByte_i/(PHT_S*PHT_D);
   	//  (i/S)%D
   	PHT_Bit_indxj:= (PHT_WordToByte_i/PHT_S) MOD PHT_D;
   
   
   	PHT_Tmp[0]:= PHT_State[PHT_Byte_indxi,PHT_Bit_indxj];
   
   	//& Wordfilter
   	If PHT_S=8 Then
   		PHT_Tmp[0]:= PHT_Tmp[0] AND 16#ff;
   	Else
   		PHT_Tmp[0]:= PHT_Tmp[0] AND 16#f;
   	End_If;
   
   	//>>(S-min(S, NoOfBits-i))
   	CASE PHT_Tmp[1] OF
   		1:
   			PHT_Tmp[0]:=PHT_Tmp[0]/2;
   		2:
   			PHT_Tmp[0]:=PHT_Tmp[0]/4;
   
   		3:
   			PHT_Tmp[0]:=PHT_Tmp[0]/8;
   		4:
   			PHT_Tmp[0]:=PHT_Tmp[0]/16;
   		5:
   			PHT_Tmp[0]:=PHT_Tmp[0]/32;
   		6:
   			PHT_Tmp[0]:=PHT_Tmp[0]/64;
   		7:
   			PHT_Tmp[0]:=PHT_Tmp[0]/128;
   		8:
   			PHT_Tmp[0]:=PHT_Tmp[0]/256;
   	End_Case;
   	PHT_WriteByte_Value:=PHT_Tmp[0];
   
   	JSR(PHOTON_WriteByte);
   
   
   
   	PHT_WordToByte_i:=PHT_WordToByte_i+PHT_S;
   
   End_While;
END_ROUTINE

ROUTINE PHOTON_WordXorByte   (* structured text *)
   (*
   void WordXorByte(byte state[D][D], const byte*str, int BitOffSet, int WordOffSet, int NoOfBits)
   {
   	int i = 0;
   	while(i < NoOfBits)
   	{
   		state[(WordOffSet+(i/S))/D][(WordOffSet+(i/S))%D] ^= GetByte(str, BitOffSet+i, min(S, NoOfBits-i))<<(S-min(S,NoOfBits-i));
   		i += S;
   	}
   }
   *)
   
   
   
   
   PHT_WordXorByte_i:=0;
   
   While PHT_WordXorByte_i<PHT_WordXorByte_NoOfBits Do
   	PHT_Byte_indxi:=  (PHT_WordXorByte_WordOffset+(PHT_WordXorByte_i/PHT_S))/PHT_D;
   	PHT_Bit_indxj:= (PHT_WordXorByte_WordOffset+(PHT_WordXorByte_i/PHT_S)) MOD PHT_D;
   
   	PHT_GetByte_BitOffSet:=PHT_WordXorByte_BitOffSet + PHT_WordXorByte_i;
   
   	//min(S,NoOfBits-i)
   	PHT_Tmp[0]:=PHT_WordXorByte_NoOfBits- PHT_WordXorByte_i;
   	if PHT_Tmp[0]> PHT_S Then
   		PHT_Tmp[0]:=PHT_S;
   	End_if;
   
   
   	PHT_GetByte_NoOfBits:=PHT_Tmp[0];
   
   	JSR(PHOTON_GetByte);
   
   	PHT_Tmp[0]:= PHT_S- PHT_GetByte_NoOfBits;
   
   	CASE PHT_Tmp[0] OF
   		1:
   			PHT_GetByte_Res:=PHT_GetByte_Res*2;
   		2:
   			PHT_GetByte_Res:=PHT_GetByte_Res*4;
   
   		3:
   			PHT_GetByte_Res:=PHT_GetByte_Res*8;
   		4:
   			PHT_GetByte_Res:=PHT_GetByte_Res*16;
   		5:
   			PHT_GetByte_Res:=PHT_GetByte_Res*32;
   		6:
   			PHT_GetByte_Res:=PHT_GetByte_Res*64;
   		7:
   			PHT_GetByte_Res:=PHT_GetByte_Res*128;
   		8:
   			PHT_GetByte_Res:=PHT_GetByte_Res*256;
   	End_Case;
   
   	If PHT_S=4 Then
   		PHT_State[PHT_Byte_indxi,PHT_Bit_indxj]:=(PHT_State[PHT_Byte_indxi,PHT_Bit_indxj] XOR PHT_GetByte_Res) AND 16#F;
   	else
   		PHT_State[PHT_Byte_indxi,PHT_Bit_indxj]:=(PHT_State[PHT_Byte_indxi,PHT_Bit_indxj] XOR PHT_GetByte_Res) AND 16#Ff;
   	End_if;
   
   
   
   
   
   
   
   	PHT_WordXorByte_i:=PHT_WordXorByte_i+PHT_S;
   End_while;
END_ROUTINE

ROUTINE PHOTON_WriteByte   (* structured text *)
   	(*
   /* ensure NoOfBits <=8 */
   void WriteByte(byte*str, byte value, int BitOffSet, int NoOfBits)
   {
   	int ByteIndex = BitOffSet >> 3;
   	int BitIndex = BitOffSet & 0x7;
   	byte localFilter = (((byte)1)<<NoOfBits) - 1;
   	value &= localFilter;
   	if(BitIndex+ NoOfBits <= 8) {
   		str[ByteIndex] &= ~(localFilter<<(8-BitIndex-NoOfBits));
   		str[ByteIndex] |= value<<(8-BitIndex-NoOfBits);
   	}
   	else {
   		u32 tmp = ((((u32) str[ByteIndex])<<8)&0xFF00) | (((u32) str[ByteIndex+1])&0xFF);
   		tmp &= ~((((u32)localFilter)&0xFF)<<(16-BitIndex-NoOfBits));
   		tmp |= (((u32)(value))&0xFF)<<(16-BitIndex-NoOfBits);
   		str[ByteIndex] = (tmp>>8)&0xFF;
   		str[ByteIndex+1] = tmp&0xFF;
   	}
   }*)
   	// ByteIndex = BitOffSet >> 3;
   	PHT_Byte_indxi:=PHT_WriteByte_BitOffset/8;
   	//BitIndex = BitOffSet & 0x7;
   	PHT_Bit_indxj:=PHT_WriteByte_BitOffset AND 16#7;
   	//localFilter = (((byte)1)<<NoOfBits) - 1;
   	PHT_WriteByte_LocalFilter:=0;
   	PHT_WriteByte_LocalFilter.[PHT_WriteByte_NoOfBits]:=1;
   	PHT_WriteByte_LocalFilter:=PHT_WriteByte_LocalFilter-1;
   
   	PHT_WriteByte_Value:= PHT_WriteByte_Value AND PHT_WriteByte_LocalFilter;
   
   	If PHT_Bit_indxj+ PHT_WriteByte_NoOfBits <=8 Then
   
   		PHT_Tmp[1]:= 8-PHT_Bit_indxj-PHT_WriteByte_NoOfBits;
   		CASE PHT_Tmp[1] OF
   			1:
   				PHT_WriteByte_LocalFilter:=PHT_WriteByte_LocalFilter*2;
   				PHT_WriteByte_Value:=PHT_WriteByte_Value*2;
   			2:
   				PHT_WriteByte_LocalFilter:=PHT_WriteByte_LocalFilter*4;
   				PHT_WriteByte_Value:=PHT_WriteByte_Value*4;
   
   			3:
   				PHT_WriteByte_LocalFilter:=PHT_WriteByte_LocalFilter*8;
   				PHT_WriteByte_Value:=PHT_WriteByte_Value*8;
   			4:
   				PHT_WriteByte_LocalFilter:=PHT_WriteByte_LocalFilter*16;
   				PHT_WriteByte_Value:=PHT_WriteByte_Value*16;
   			5:
   				PHT_WriteByte_LocalFilter:=PHT_WriteByte_LocalFilter*32;
   				PHT_WriteByte_Value:=PHT_WriteByte_Value*32;
   			6:
   				PHT_WriteByte_LocalFilter:=PHT_WriteByte_LocalFilter*64;
   				PHT_WriteByte_Value:=PHT_WriteByte_Value*64;
   			7:
   				PHT_WriteByte_LocalFilter:=PHT_WriteByte_LocalFilter*128;
   				PHT_WriteByte_Value:=PHT_WriteByte_Value*128;
   			8:
   				PHT_WriteByte_LocalFilter:=PHT_WriteByte_LocalFilter*256;
   				PHT_WriteByte_Value:=PHT_WriteByte_Value*256;
   		End_Case;
   		//Digest[ByteIndex] &= ~(localFilter<<(8-BitIndex-NoOfBits));
   		//Digest[ByteIndex] |= value<<(8-BitIndex-NoOfBits
   			PHT_WriteByte_LocalFilter:=(NOT PHT_WriteByte_LocalFilter) ;
   			PHT_Digest[PHT_Byte_indxi]:= PHT_Digest[PHT_Byte_indxi] AND PHT_WriteByte_LocalFilter;
   			PHT_Digest[PHT_Byte_indxi]:= PHT_Digest[PHT_Byte_indxi] OR PHT_WriteByte_Value;
   
   
   	Else
   		//u32 tmp = ((((u32) str[ByteIndex])<<8)&0xFF00) | (((u32) str[ByteIndex+1])&0xFF);
   		//tmp &= ~((((u32)localFilter)&0xFF)<<(16-BitIndex-NoOfBits));
   		//tmp |= (((u32)(value))&0xFF)<<(16-BitIndex-NoOfBits);
   
   		PHT_Tmp[0]:= ((PHT_Digest[PHT_Byte_indxi]*256) AND 16#FF00) OR (PHT_Digest[PHT_Byte_indxi+1] AND 16#FF);
   		PHT_Tmp[1]:= 16-PHT_Bit_indxj-PHT_WriteByte_NoOfBits;
   		Case PHT_Tmp[1] Of
   				1:
   					PHT_Tmp[0]:=PHT_Tmp[0] AND (NOT ((PHT_WriteByte_LocalFilter AND 16#FF)* 2));
   					PHT_Tmp[0]:=PHT_Tmp[0] OR ((PHT_WriteByte_Value AND 16#FF)* 2);
   				2:
   					PHT_Tmp[0]:=PHT_Tmp[0] AND (NOT ((PHT_WriteByte_LocalFilter AND 16#FF)* 4));
   					PHT_Tmp[0]:=PHT_Tmp[0] OR ((PHT_WriteByte_Value AND 16#FF)* 4);
   				3:
   					PHT_Tmp[0]:=PHT_Tmp[0] AND (NOT ((PHT_WriteByte_LocalFilter AND 16#FF)* 8));
   					PHT_Tmp[0]:=PHT_Tmp[0] OR ((PHT_WriteByte_Value AND 16#FF)* 8);
   				4:
   					PHT_Tmp[0]:=PHT_Tmp[0] AND (NOT ((PHT_WriteByte_LocalFilter AND 16#FF)* 16));
   					PHT_Tmp[0]:=PHT_Tmp[0] OR ((PHT_WriteByte_Value AND 16#FF)* 16);
   				5:
   					PHT_Tmp[0]:=PHT_Tmp[0] AND (NOT ((PHT_WriteByte_LocalFilter AND 16#FF)* 32));
   					PHT_Tmp[0]:=PHT_Tmp[0] OR ((PHT_WriteByte_Value AND 16#FF)* 32);
   				6:
   					PHT_Tmp[0]:=PHT_Tmp[0] AND (NOT ((PHT_WriteByte_LocalFilter AND 16#FF)* 64));
   					PHT_Tmp[0]:=PHT_Tmp[0] OR ((PHT_WriteByte_Value AND 16#FF)* 64);
   				7:
   					PHT_Tmp[0]:=PHT_Tmp[0] AND (NOT ((PHT_WriteByte_LocalFilter AND 16#FF)* 128));
   					PHT_Tmp[0]:=PHT_Tmp[0] OR ((PHT_WriteByte_Value AND 16#FF)* 128);
   				8:
   					PHT_Tmp[0]:=PHT_Tmp[0] AND (NOT ((PHT_WriteByte_LocalFilter AND 16#FF)* 256));
   					PHT_Tmp[0]:=PHT_Tmp[0] OR ((PHT_WriteByte_Value AND 16#FF)* 256);
   				9:
   					PHT_Tmp[0]:=PHT_Tmp[0] AND (NOT ((PHT_WriteByte_LocalFilter AND 16#FF)* 512));
   					PHT_Tmp[0]:=PHT_Tmp[0] OR ((PHT_WriteByte_Value AND 16#FF)* 512);
   				10:
   					PHT_Tmp[0]:=PHT_Tmp[0] AND (NOT ((PHT_WriteByte_LocalFilter AND 16#FF)* 1024));
   					PHT_Tmp[0]:=PHT_Tmp[0] OR ((PHT_WriteByte_Value AND 16#FF)* 1024);
   				11:
   					PHT_Tmp[0]:=PHT_Tmp[0] AND (NOT ((PHT_WriteByte_LocalFilter AND 16#FF)* 2048));
   					PHT_Tmp[0]:=PHT_Tmp[0] OR ((PHT_WriteByte_Value AND 16#FF)* 2048);
   				12:
   					PHT_Tmp[0]:=PHT_Tmp[0] AND (NOT ((PHT_WriteByte_LocalFilter AND 16#FF)* 4096));
   					PHT_Tmp[0]:=PHT_Tmp[0] OR ((PHT_WriteByte_Value AND 16#FF)* 4096);
   				13:
   					PHT_Tmp[0]:=PHT_Tmp[0] AND (NOT ((PHT_WriteByte_LocalFilter AND 16#FF)* 8192));
   					PHT_Tmp[0]:=PHT_Tmp[0] OR ((PHT_WriteByte_Value AND 16#FF)* 8192);
   				14:
   					PHT_Tmp[0]:=PHT_Tmp[0] AND (NOT ((PHT_WriteByte_LocalFilter AND 16#FF)* 16384));
   					PHT_Tmp[0]:=PHT_Tmp[0] OR ((PHT_WriteByte_Value AND 16#FF)* 16384);
   				15:
   					PHT_Tmp[0]:=PHT_Tmp[0] AND (NOT ((PHT_WriteByte_LocalFilter AND 16#FF)* 32768));
   					PHT_Tmp[0]:=PHT_Tmp[0] OR ((PHT_WriteByte_Value AND 16#FF)* 32768);
   				16:
   					PHT_Tmp[0]:=PHT_Tmp[0] AND (NOT ((PHT_WriteByte_LocalFilter AND 16#FF)* 65536));
   					PHT_Tmp[0]:=PHT_Tmp[0] OR ((PHT_WriteByte_Value AND 16#FF)* 65536);
   
   
   
   
   		End_Case;
   		//str[ByteIndex] = (tmp>>8)&0xFF;
   		//str[ByteIndex+1] = tmp&0xFF;
   
   
   		PHT_Digest[PHT_Byte_indxi]:= (PHT_Tmp[0]/256)AND 16#FF;
   		PHT_Digest[PHT_Byte_indxi+1]:=PHT_Tmp[0] AND 16#FF;
   
   
   	End_if;
   
END_ROUTINE
END_PROGRAM
